LIN {X -112.913,Y -21.431,Z -236.404,A -90.000,B 90.000,C 0.000} C_DIS
LIN {X -101.773,Y -21.431,Z -228.606,A -90.000,B 90.000,C 0.000} C_DIS
LIN {X -97.009,Y -21.431,Z -225.268,A -90.000,B 90.000,C 0.000} C_DIS
LIN {X -92.221,Y -21.431,Z -221.963,A -90.000,B 90.000,C 0.000} C_DIS
LIN {X -87.411,Y -21.431,Z -218.691,A -90.000,B 90.000,C 0.000} C_DIS
LIN {X -82.578,Y -21.431,Z -215.452,A -90.000,B 90.000,C 0.000} C_DIS
LIN {X -77.723,Y -21.431,Z -212.248,A -90.000,B 90.000,C 0.000} C_DIS
LIN {X -69.739,Y -21.431,Z -206.990,A -90.000,B 90.000,C 0.000} C_DIS
LIN {X -65.801,Y -21.431,Z -204.457,A -90.000,B 90.000,C 0.000} C_DIS
LIN {X -61.895,Y -21.431,Z -201.875,A -90.000,B 90.000,C 0.000} C_DIS
LIN {X -58.021,Y -21.431,Z -199.246,A -90.000,B 90.000,C 0.000} C_DIS
LIN {X -54.179,Y -21.431,Z -196.569,A -90.000,B 90.000,C 0.000} C_DIS
LIN {X -50.371,Y -21.431,Z -193.845,A -90.000,B 90.000,C 0.000} C_DIS
LIN {X -46.597,Y -21.431,Z -191.074,A -90.000,B 90.000,C 0.000} C_DIS
LIN {X -42.857,Y -21.431,Z -188.257,A -90.000,B 90.000,C 0.000} C_DIS
LIN {X -39.152,Y -21.431,Z -185.394,A -90.000,B 90.000,C 0.000} C_DIS
LIN {X -35.482,Y -21.431,Z -182.486,A -90.000,B 90.000,C 0.000} C_DIS
LIN {X -33.831,Y -21.431,Z -181.236,A -90.000,B 90.000,C 0.000} C_DIS
LIN {X -32.219,Y -21.431,Z -179.937,A -90.000,B 90.000,C 0.000} C_DIS
LIN {X -30.645,Y -21.431,Z -178.592,A -90.000,B 90.000,C 0.000} C_DIS
LIN {X -29.112,Y -21.431,Z -177.200,A -90.000,B 90.000,C 0.000} C_DIS
LIN {X -27.621,Y -21.431,Z -175.763,A -90.000,B 90.000,C 0.000} C_DIS
LIN {X -26.173,Y -21.431,Z -174.283,A -90.000,B 90.000,C 0.000} C_DIS
LIN {X -24.770,Y -21.431,Z -172.761,A -90.000,B 90.000,C 0.000} C_DIS
LIN {X -23.815,Y -21.431,Z -171.758,A -90.000,B 90.000,C 0.000} C_DIS
LIN {X -22.906,Y -21.431,Z -170.713,A -90.000,B 90.000,C 0.000} C_DIS
LIN {X -22.045,Y -21.431,Z -169.628,A -90.000,B 90.000,C 0.000} C_DIS
LIN {X -21.234,Y -21.431,Z -168.506,A -90.000,B 90.000,C 0.000} C_DIS
LIN {X -20.473,Y -21.431,Z -167.349,A -90.000,B 90.000,C 0.000} C_DIS
LIN {X -19.766,Y -21.431,Z -166.158,A -90.000,B 90.000,C 0.000} C_DIS
LIN {X -19.112,Y -21.431,Z -164.937,A -90.000,B 90.000,C 0.000} C_DIS
LIN {X -18.514,Y -21.431,Z -163.688,A -90.000,B 90.000,C 0.000} C_DIS
LIN {X -18.456,Y -21.431,Z -163.541,A -90.000,B 90.000,C 0.000} C_DIS
LIN {X -19.036,Y -21.431,Z -162.884,A -90.000,B 90.000,C 0.000} C_DIS
LIN {X -19.116,Y -21.431,Z -162.777,A -90.000,B 90.000,C 0.000} C_DIS
LIN {X -19.886,Y -21.431,Z -161.971,A -90.000,B 90.000,C 0.000} C_DIS
LIN {X -20.688,Y -21.431,Z -161.196,A -90.000,B 90.000,C 0.000} C_DIS
LIN {X -23.607,Y -21.431,Z -158.546,A -90.000,B 90.000,C 0.000} C_DIS
LIN {X -26.501,Y -21.431,Z -155.871,A -90.000,B 90.000,C 0.000} C_DIS
LIN {X -29.372,Y -21.431,Z -153.169,A -90.000,B 90.000,C 0.000} C_DIS
LIN {X -30.672,Y -21.431,Z -151.944,A -90.000,B 90.000,C 0.000} C_DIS
LIN {X -31.934,Y -21.431,Z -150.679,A -90.000,B 90.000,C 0.000} C_DIS
LIN {X -33.157,Y -21.431,Z -149.377,A -90.000,B 90.000,C 0.000} C_DIS
LIN {X -34.339,Y -21.431,Z -148.039,A -90.000,B 90.000,C 0.000} C_DIS
LIN {X -35.481,Y -21.431,Z -146.664,A -90.000,B 90.000,C 0.000} C_DIS
LIN {X -36.579,Y -21.431,Z -145.256,A -90.000,B 90.000,C 0.000} C_DIS
LIN {X -37.635,Y -21.431,Z -143.815,A -90.000,B 90.000,C 0.000} C_DIS
LIN {X -38.762,Y -21.431,Z -142.053,A -90.000,B 90.000,C 0.000} C_DIS
LIN {X -39.842,Y -21.431,Z -140.263,A -90.000,B 90.000,C 0.000} C_DIS
LIN {X -40.874,Y -21.431,Z -138.445,A -90.000,B 90.000,C 0.000} C_DIS
LIN {X -41.859,Y -21.431,Z -136.600,A -90.000,B 90.000,C 0.000} C_DIS
LIN {X -42.796,Y -21.431,Z -134.730,A -90.000,B 90.000,C 0.000} C_DIS
LIN {X -43.682,Y -21.431,Z -132.837,A -90.000,B 90.000,C 0.000} C_DIS
LIN {X -44.519,Y -21.431,Z -130.920,A -90.000,B 90.000,C 0.000} C_DIS
LIN {X -45.306,Y -21.431,Z -128.983,A -90.000,B 90.000,C 0.000} C_DIS
LIN {X -45.631,Y -21.431,Z -127.972,A -90.000,B 90.000,C 0.000} C_DIS
LIN {X -46.007,Y -21.431,Z -126.979,A -90.000,B 90.000,C 0.000} C_DIS
LIN {X -46.431,Y -21.431,Z -126.006,A -90.000,B 90.000,C 0.000} C_DIS
LIN {X -46.904,Y -21.431,Z -125.055,A -90.000,B 90.000,C 0.000} C_DIS
LIN {X -47.424,Y -21.431,Z -124.129,A -90.000,B 90.000,C 0.000} C_DIS
LIN {X -47.989,Y -21.431,Z -123.230,A -90.000,B 90.000,C 0.000} C_DIS
LIN {X -50.279,Y -21.431,Z -120.489,A -90.000,B 90.000,C 0.000} C_DIS
LIN {X -52.532,Y -21.431,Z -117.717,A -90.000,B 90.000,C 0.000} C_DIS
LIN {X -54.746,Y -21.431,Z -114.914,A -90.000,B 90.000,C 0.000} C_DIS
LIN {X -56.921,Y -21.431,Z -112.081,A -90.000,B 90.000,C 0.000} C_DIS
LIN {X -59.058,Y -21.431,Z -109.218,A -90.000,B 90.000,C 0.000} C_DIS
LIN {X -61.154,Y -21.431,Z -106.326,A -90.000,B 90.000,C 0.000} C_DIS
LIN {X -62.757,Y -21.431,Z -104.098,A -90.000,B 90.000,C 0.000} C_DIS
LIN {X -64.383,Y -21.431,Z -101.888,A -90.000,B 90.000,C 0.000} C_DIS
LIN {X -65.729,Y -21.431,Z -100.052,A -90.000,B 90.000,C 0.000} C_DIS
LIN {X -67.124,Y -21.431,Z -98.251,A -90.000,B 90.000,C 0.000} C_DIS
LIN {X -68.566,Y -21.431,Z -96.489,A -90.000,B 90.000,C 0.000} C_DIS
LIN {X -70.054,Y -21.431,Z -94.765,A -90.000,B 90.000,C 0.000} C_DIS
LIN {X -71.588,Y -21.431,Z -93.082,A -90.000,B 90.000,C 0.000} C_DIS
LIN {X -73.165,Y -21.431,Z -91.439,A -90.000,B 90.000,C 0.000} C_DIS
LIN {X -74.786,Y -21.431,Z -89.839,A -90.000,B 90.000,C 0.000} C_DIS
LIN {X -76.448,Y -21.431,Z -88.283,A -90.000,B 90.000,C 0.000} C_DIS
LIN {X -76.915,Y -21.431,Z -87.802,A -90.000,B 90.000,C 0.000} C_DIS
LIN {X -77.417,Y -21.431,Z -87.357,A -90.000,B 90.000,C 0.000} C_DIS
LIN {X -77.950,Y -21.431,Z -86.950,A -90.000,B 90.000,C 0.000} C_DIS
LIN {X -78.511,Y -21.431,Z -86.584,A -90.000,B 90.000,C 0.000} C_DIS
LIN {X -79.099,Y -21.431,Z -86.260,A -90.000,B 90.000,C 0.000} C_DIS
LIN {X -79.708,Y -21.431,Z -85.980,A -90.000,B 90.000,C 0.000} C_DIS
LIN {X -81.105,Y -21.431,Z -85.489,A -90.000,B 90.000,C 0.000} C_DIS
LIN {X -82.479,Y -21.431,Z -84.936,A -90.000,B 90.000,C 0.000} C_DIS
LIN {X -83.828,Y -21.431,Z -84.323,A -90.000,B 90.000,C 0.000} C_DIS
LIN {X -85.147,Y -21.431,Z -83.651,A -90.000,B 90.000,C 0.000} C_DIS
LIN {X -86.436,Y -21.431,Z -82.921,A -90.000,B 90.000,C 0.000} C_DIS
LIN {X -87.691,Y -21.431,Z -82.134,A -90.000,B 90.000,C 0.000} C_DIS
LIN {X -88.909,Y -21.431,Z -81.292,A -90.000,B 90.000,C 0.000} C_DIS
LIN {X -90.090,Y -21.431,Z -80.398,A -90.000,B 90.000,C 0.000} C_DIS
LIN {X -90.244,Y -21.431,Z -80.288,A -90.000,B 90.000,C 0.000} C_DIS
LIN {X -92.608,Y -21.431,Z -78.373,A -90.000,B 90.000,C 0.000} C_DIS
LIN {X -94.982,Y -21.431,Z -76.470,A -90.000,B 90.000,C 0.000} C_DIS
LIN {X -96.724,Y -21.431,Z -75.460,A -90.000,B 90.000,C 0.000} C_DIS
LIN {X -98.431,Y -21.431,Z -74.393,A -90.000,B 90.000,C 0.000} C_DIS
LIN {X -100.102,Y -21.431,Z -73.269,A -90.000,B 90.000,C 0.000} C_DIS
LIN {X -101.734,Y -21.431,Z -72.091,A -90.000,B 90.000,C 0.000} C_DIS
LIN {X -103.327,Y -21.431,Z -70.859,A -90.000,B 90.000,C 0.000} C_DIS
LIN {X -104.877,Y -21.431,Z -69.575,A -90.000,B 90.000,C 0.000} C_DIS
LIN {X -106.385,Y -21.431,Z -68.240,A -90.000,B 90.000,C 0.000} C_DIS
LIN {X -107.846,Y -21.431,Z -66.856,A -90.000,B 90.000,C 0.000} C_DIS
LIN {X -109.262,Y -21.431,Z -65.424,A -90.000,B 90.000,C 0.000} C_DIS
LIN {X -110.628,Y -21.431,Z -63.945,A -90.000,B 90.000,C 0.000} C_DIS
LIN {X -111.945,Y -21.431,Z -62.422,A -90.000,B 90.000,C 0.000} C_DIS
LIN {X -112.631,Y -21.431,Z -61.641,A -90.000,B 90.000,C 0.000} C_DIS
LIN {X -113.269,Y -21.431,Z -60.819,A -90.000,B 90.000,C 0.000} C_DIS
LIN {X -113.855,Y -21.431,Z -59.960,A -90.000,B 90.000,C 0.000} C_DIS
LIN {X -114.388,Y -21.431,Z -59.066,A -90.000,B 90.000,C 0.000} C_DIS
LIN {X -114.865,Y -21.431,Z -58.142,A -90.000,B 90.000,C 0.000} C_DIS
LIN {X -115.284,Y -21.431,Z -57.190,A -90.000,B 90.000,C 0.000} C_DIS
LIN {X -115.645,Y -21.431,Z -56.215,A -90.000,B 90.000,C 0.000} C_DIS
LIN {X -115.945,Y -21.431,Z -55.219,A -90.000,B 90.000,C 0.000} C_DIS
LIN {X -116.219,Y -21.431,Z -54.365,A -90.000,B 90.000,C 0.000} C_DIS
LIN {X -116.430,Y -21.431,Z -53.494,A -90.000,B 90.000,C 0.000} C_DIS
LIN {X -116.579,Y -21.431,Z -52.609,A -90.000,B 90.000,C 0.000} C_DIS
LIN {X -116.664,Y -21.431,Z -51.717,A -90.000,B 90.000,C 0.000} C_DIS
LIN {X -116.684,Y -21.431,Z -50.820,A -90.000,B 90.000,C 0.000} C_DIS
LIN {X -116.640,Y -21.431,Z -49.924,A -90.000,B 90.000,C 0.000} C_DIS
LIN {X -116.532,Y -21.431,Z -49.034,A -90.000,B 90.000,C 0.000} C_DIS
LIN {X -116.361,Y -21.431,Z -48.154,A -90.000,B 90.000,C 0.000} C_DIS
LIN {X -116.729,Y -21.431,Z -47.203,A -90.000,B 90.000,C 0.000} C_DIS
LIN {X -117.034,Y -21.431,Z -46.230,A -90.000,B 90.000,C 0.000} C_DIS
LIN {X -117.276,Y -21.431,Z -45.239,A -90.000,B 90.000,C 0.000} C_DIS
LIN {X -117.453,Y -21.431,Z -44.235,A -90.000,B 90.000,C 0.000} C_DIS
LIN {X -117.565,Y -21.431,Z -43.221,A -90.000,B 90.000,C 0.000} C_DIS
LIN {X -117.611,Y -21.431,Z -42.203,A -90.000,B 90.000,C 0.000} C_DIS
LIN {X -117.592,Y -21.431,Z -41.183,A -90.000,B 90.000,C 0.000} C_DIS
LIN {X -117.506,Y -21.431,Z -40.167,A -90.000,B 90.000,C 0.000} C_DIS
LIN {X -117.481,Y -21.431,Z -39.998,A -90.000,B 90.000,C 0.000} C_DIS
LIN {X -117.325,Y -21.431,Z -39.111,A -90.000,B 90.000,C 0.000} C_DIS
LIN {X -117.112,Y -21.431,Z -38.236,A -90.000,B 90.000,C 0.000} C_DIS
LIN {X -116.843,Y -21.431,Z -37.377,A -90.000,B 90.000,C 0.000} C_DIS
LIN {X -116.518,Y -21.431,Z -36.537,A -90.000,B 90.000,C 0.000} C_DIS
LIN {X -116.140,Y -21.431,Z -35.720,A -90.000,B 90.000,C 0.000} C_DIS
LIN {X -115.709,Y -21.431,Z -34.929,A -90.000,B 90.000,C 0.000} C_DIS
LIN {X -115.632,Y -21.431,Z -34.808,A -90.000,B 90.000,C 0.000} C_DIS
LIN {X -115.195,Y -21.431,Z -34.136,A -90.000,B 90.000,C 0.000} C_DIS
LIN {X -114.713,Y -21.431,Z -33.495,A -90.000,B 90.000,C 0.000} C_DIS
LIN {X -114.188,Y -21.431,Z -32.888,A -90.000,B 90.000,C 0.000} C_DIS
LIN {X -113.624,Y -21.431,Z -32.318,A -90.000,B 90.000,C 0.000} C_DIS
LIN {X -113.490,Y -21.431,Z -32.194,A -90.000,B 90.000,C 0.000} C_DIS
LIN {X -112.360,Y -21.431,Z -31.268,A -90.000,B 90.000,C 0.000} C_DIS
LIN {X -112.270,Y -21.431,Z -31.206,A -90.000,B 90.000,C 0.000} C_DIS
LIN {X -111.804,Y -21.431,Z -30.880,A -90.000,B 90.000,C 0.000} C_DIS
LIN {X -111.318,Y -21.431,Z -30.585,A -90.000,B 90.000,C 0.000} C_DIS
LIN {X -110.813,Y -21.431,Z -30.324,A -90.000,B 90.000,C 0.000} C_DIS
LIN {X -110.292,Y -21.431,Z -30.095,A -90.000,B 90.000,C 0.000} C_DIS
LIN {X -109.345,Y -21.431,Z -29.251,A -90.000,B 90.000,C 0.000} C_DIS
LIN {X -108.357,Y -21.431,Z -28.456,A -90.000,B 90.000,C 0.000} C_DIS
LIN {X -107.331,Y -21.431,Z -27.711,A -90.000,B 90.000,C 0.000} C_DIS
LIN {X -106.268,Y -21.431,Z -27.018,A -90.000,B 90.000,C 0.000} C_DIS
LIN {X -105.172,Y -21.431,Z -26.380,A -90.000,B 90.000,C 0.000} C_DIS
LIN {X -104.800,Y -21.431,Z -25.659,A -90.000,B 90.000,C 0.000} C_DIS
LIN {X -104.385,Y -21.431,Z -24.961,A -90.000,B 90.000,C 0.000} C_DIS
LIN {X -103.928,Y -21.431,Z -24.289,A -90.000,B 90.000,C 0.000} C_DIS
LIN {X -103.432,Y -21.431,Z -23.647,A -90.000,B 90.000,C 0.000} C_DIS
LIN {X -102.917,Y -21.431,Z -22.919,A -90.000,B 90.000,C 0.000} C_DIS
LIN {X -102.353,Y -21.431,Z -22.229,A -90.000,B 90.000,C 0.000} C_DIS
LIN {X -101.741,Y -21.431,Z -21.581,A -90.000,B 90.000,C 0.000} C_DIS
LIN {X -101.084,Y -21.431,Z -20.977,A -90.000,B 90.000,C 0.000} C_DIS
LIN {X -100.387,Y -21.431,Z -20.422,A -90.000,B 90.000,C 0.000} C_DIS
LIN {X -99.653,Y -21.431,Z -19.917,A -90.000,B 90.000,C 0.000} C_DIS
LIN {X -98.884,Y -21.431,Z -19.465,A -90.000,B 90.000,C 0.000} C_DIS
LIN {X -98.086,Y -21.431,Z -19.068,A -90.000,B 90.000,C 0.000} C_DIS
LIN {X -97.261,Y -21.431,Z -18.729,A -90.000,B 90.000,C 0.000} C_DIS
LIN {X -96.126,Y -21.431,Z -18.440,A -90.000,B 90.000,C 0.000} C_DIS
LIN {X -94.976,Y -21.431,Z -18.214,A -90.000,B 90.000,C 0.000} C_DIS
LIN {X -93.816,Y -21.431,Z -18.051,A -90.000,B 90.000,C 0.000} C_DIS
LIN {X -92.649,Y -21.431,Z -17.952,A -90.000,B 90.000,C 0.000} C_DIS
LIN {X -91.478,Y -21.431,Z -17.916,A -90.000,B 90.000,C 0.000} C_DIS
LIN {X -91.153,Y -21.431,Z -17.123,A -90.000,B 90.000,C 0.000} C_DIS
LIN {X -90.777,Y -21.431,Z -16.352,A -90.000,B 90.000,C 0.000} C_DIS
LIN {X -90.350,Y -21.431,Z -15.609,A -90.000,B 90.000,C 0.000} C_DIS
LIN {X -89.876,Y -21.431,Z -14.895,A -90.000,B 90.000,C 0.000} C_DIS
LIN {X -89.355,Y -21.431,Z -14.214,A -90.000,B 90.000,C 0.000} C_DIS
LIN {X -88.791,Y -21.431,Z -13.568,A -90.000,B 90.000,C 0.000} C_DIS
LIN {X -88.035,Y -21.431,Z -12.875,A -90.000,B 90.000,C 0.000} C_DIS
LIN {X -87.234,Y -21.431,Z -12.236,A -90.000,B 90.000,C 0.000} C_DIS
LIN {X -86.391,Y -21.431,Z -11.651,A -90.000,B 90.000,C 0.000} C_DIS
LIN {X -85.512,Y -21.431,Z -11.125,A -90.000,B 90.000,C 0.000} C_DIS
LIN {X -84.598,Y -21.431,Z -10.660,A -90.000,B 90.000,C 0.000} C_DIS
LIN {X -83.655,Y -21.431,Z -10.257,A -90.000,B 90.000,C 0.000} C_DIS
LIN {X -82.687,Y -21.431,Z -9.919,A -90.000,B 90.000,C 0.000} C_DIS
LIN {X -81.699,Y -21.431,Z -9.647,A -90.000,B 90.000,C 0.000} C_DIS
LIN {X -80.694,Y -21.431,Z -9.442,A -90.000,B 90.000,C 0.000} C_DIS
LIN {X -79.678,Y -21.431,Z -9.306,A -90.000,B 90.000,C 0.000} C_DIS
LIN {X -78.655,Y -21.431,Z -9.238,A -90.000,B 90.000,C 0.000} C_DIS
LIN {X -77.406,Y -21.431,Z -9.311,A -90.000,B 90.000,C 0.000} C_DIS
LIN {X -76.163,Y -21.431,Z -9.451,A -90.000,B 90.000,C 0.000} C_DIS
LIN {X -74.929,Y -21.431,Z -9.660,A -90.000,B 90.000,C 0.000} C_DIS
LIN {X -73.709,Y -21.431,Z -9.935,A -90.000,B 90.000,C 0.000} C_DIS
LIN {X -72.505,Y -21.431,Z -10.276,A -90.000,B 90.000,C 0.000} C_DIS
LIN {X -71.322,Y -21.431,Z -10.683,A -90.000,B 90.000,C 0.000} C_DIS
LIN {X -70.163,Y -21.431,Z -11.153,A -90.000,B 90.000,C 0.000} C_DIS
LIN {X -69.031,Y -21.431,Z -11.687,A -90.000,B 90.000,C 0.000} C_DIS
LIN {X -67.874,Y -21.431,Z -12.293,A -90.000,B 90.000,C 0.000} C_DIS
LIN {X -66.751,Y -21.431,Z -12.959,A -90.000,B 90.000,C 0.000} C_DIS
LIN {X -65.664,Y -21.431,Z -13.684,A -90.000,B 90.000,C 0.000} C_DIS
LIN {X -64.617,Y -21.431,Z -14.465,A -90.000,B 90.000,C 0.000} C_DIS
LIN {X -63.613,Y -21.431,Z -15.300,A -90.000,B 90.000,C 0.000} C_DIS
LIN {X -62.655,Y -21.431,Z -16.188,A -90.000,B 90.000,C 0.000} C_DIS
LIN {X -61.745,Y -21.431,Z -17.124,A -90.000,B 90.000,C 0.000} C_DIS
LIN {X -60.885,Y -21.431,Z -18.107,A -90.000,B 90.000,C 0.000} C_DIS
LIN {X -60.078,Y -21.431,Z -19.135,A -90.000,B 90.000,C 0.000} C_DIS
LIN {X -59.327,Y -21.431,Z -20.203,A -90.000,B 90.000,C 0.000} C_DIS
LIN {X -58.595,Y -21.431,Z -21.635,A -90.000,B 90.000,C 0.000} C_DIS
LIN {X -57.857,Y -21.431,Z -23.063,A -90.000,B 90.000,C 0.000} C_DIS
LIN {X -57.794,Y -21.431,Z -23.212,A -90.000,B 90.000,C 0.000} C_DIS
LIN {X -56.492,Y -21.431,Z -23.608,A -90.000,B 90.000,C 0.000} C_DIS
LIN {X -55.174,Y -21.431,Z -23.948,A -90.000,B 90.000,C 0.000} C_DIS
LIN {X -53.842,Y -21.431,Z -24.230,A -90.000,B 90.000,C 0.000} C_DIS
LIN {X -52.500,Y -21.431,Z -24.455,A -90.000,B 90.000,C 0.000} C_DIS
LIN {X -51.149,Y -21.431,Z -24.621,A -90.000,B 90.000,C 0.000} C_DIS
LIN {X -49.792,Y -21.431,Z -24.728,A -90.000,B 90.000,C 0.000} C_DIS
LIN {X -49.617,Y -21.431,Z -24.736,A -90.000,B 90.000,C 0.000} C_DIS
LIN {X -48.809,Y -21.431,Z -24.706,A -90.000,B 90.000,C 0.000} C_DIS
LIN {X -48.001,Y -21.431,Z -24.720,A -90.000,B 90.000,C 0.000} C_DIS
LIN {X -47.195,Y -21.431,Z -24.779,A -90.000,B 90.000,C 0.000} C_DIS
LIN {X -46.393,Y -21.431,Z -24.883,A -90.000,B 90.000,C 0.000} C_DIS
LIN {X -43.339,Y -21.431,Z -24.939,A -90.000,B 90.000,C 0.000} C_DIS
LIN {X -40.286,Y -21.431,Z -25.061,A -90.000,B 90.000,C 0.000} C_DIS
LIN {X -37.237,Y -21.431,Z -25.249,A -90.000,B 90.000,C 0.000} C_DIS
LIN {X -34.193,Y -21.431,Z -25.503,A -90.000,B 90.000,C 0.000} C_DIS
LIN {X -31.155,Y -21.431,Z -25.823,A -90.000,B 90.000,C 0.000} C_DIS
LIN {X -28.125,Y -21.431,Z -26.209,A -90.000,B 90.000,C 0.000} C_DIS
LIN {X -25.104,Y -21.431,Z -26.660,A -90.000,B 90.000,C 0.000} C_DIS
LIN {X -22.093,Y -21.431,Z -27.176,A -90.000,B 90.000,C 0.000} C_DIS
LIN {X -19.094,Y -21.431,Z -27.758,A -90.000,B 90.000,C 0.000} C_DIS
LIN {X -16.108,Y -21.431,Z -28.404,A -90.000,B 90.000,C 0.000} C_DIS
LIN {X -13.137,Y -21.431,Z -29.114,A -90.000,B 90.000,C 0.000} C_DIS
LIN {X -10.182,Y -21.431,Z -29.889,A -90.000,B 90.000,C 0.000} C_DIS
LIN {X -7.245,Y -21.431,Z -30.728,A -90.000,B 90.000,C 0.000} C_DIS
LIN {X -6.078,Y -21.431,Z -31.125,A -90.000,B 90.000,C 0.000} C_DIS
LIN {X -4.894,Y -21.431,Z -31.466,A -90.000,B 90.000,C 0.000} C_DIS
LIN {X -3.694,Y -21.431,Z -31.750,A -90.000,B 90.000,C 0.000} C_DIS
LIN {X -2.482,Y -21.431,Z -31.977,A -90.000,B 90.000,C 0.000} C_DIS
LIN {X -1.261,Y -21.431,Z -32.145,A -90.000,B 90.000,C 0.000} C_DIS
LIN {X -0.034,Y -21.431,Z -32.255,A -90.000,B 90.000,C 0.000} C_DIS
LIN {X 1.198,Y -21.431,Z -32.305,A -90.000,B 90.000,C 0.000} C_DIS
LIN {X 3.136,Y -21.431,Z -32.301,A -90.000,B 90.000,C 0.000} C_DIS
LIN {X 5.073,Y -21.431,Z -32.346,A -90.000,B 90.000,C 0.000} C_DIS
LIN {X 7.009,Y -21.431,Z -32.440,A -90.000,B 90.000,C 0.000} C_DIS
LIN {X 8.942,Y -21.431,Z -32.584,A -90.000,B 90.000,C 0.000} C_DIS
LIN {X 10.870,Y -21.431,Z -32.776,A -90.000,B 90.000,C 0.000} C_DIS
LIN {X 12.793,Y -21.431,Z -33.017,A -90.000,B 90.000,C 0.000} C_DIS
LIN {X 14.148,Y -21.431,Z -33.216,A -90.000,B 90.000,C 0.000} C_DIS
LIN {X 15.510,Y -21.431,Z -33.360,A -90.000,B 90.000,C 0.000} C_DIS
LIN {X 16.877,Y -21.431,Z -33.450,A -90.000,B 90.000,C 0.000} C_DIS
LIN {X 18.246,Y -21.431,Z -33.486,A -90.000,B 90.000,C 0.000} C_DIS
LIN {X 19.616,Y -21.431,Z -33.466,A -90.000,B 90.000,C 0.000} C_DIS
LIN {X 20.983,Y -21.431,Z -33.392,A -90.000,B 90.000,C 0.000} C_DIS
LIN {X 22.347,Y -21.431,Z -33.264,A -90.000,B 90.000,C 0.000} C_DIS
LIN {X 25.111,Y -21.431,Z -32.751,A -90.000,B 90.000,C 0.000} C_DIS
LIN {X 27.884,Y -21.431,Z -32.288,A -90.000,B 90.000,C 0.000} C_DIS
LIN {X 30.665,Y -21.431,Z -31.876,A -90.000,B 90.000,C 0.000} C_DIS
LIN {X 33.453,Y -21.431,Z -31.514,A -90.000,B 90.000,C 0.000} C_DIS
LIN {X 35.088,Y -21.431,Z -31.430,A -90.000,B 90.000,C 0.000} C_DIS
LIN {X 36.726,Y -21.431,Z -31.411,A -90.000,B 90.000,C 0.000} C_DIS
LIN {X 38.362,Y -21.431,Z -31.456,A -90.000,B 90.000,C 0.000} C_DIS
LIN {X 39.996,Y -21.431,Z -31.566,A -90.000,B 90.000,C 0.000} C_DIS
LIN {X 41.624,Y -21.431,Z -31.741,A -90.000,B 90.000,C 0.000} C_DIS
LIN {X 43.244,Y -21.431,Z -31.980,A -90.000,B 90.000,C 0.000} C_DIS
LIN {X 44.853,Y -21.431,Z -32.283,A -90.000,B 90.000,C 0.000} C_DIS
LIN {X 46.520,Y -21.431,Z -32.778,A -90.000,B 90.000,C 0.000} C_DIS
LIN {X 48.167,Y -21.431,Z -33.333,A -90.000,B 90.000,C 0.000} C_DIS
LIN {X 49.794,Y -21.431,Z -33.947,A -90.000,B 90.000,C 0.000} C_DIS
LIN {X 51.397,Y -21.431,Z -34.619,A -90.000,B 90.000,C 0.000} C_DIS
LIN {X 52.976,Y -21.431,Z -35.348,A -90.000,B 90.000,C 0.000} C_DIS
LIN {X 54.527,Y -21.431,Z -36.133,A -90.000,B 90.000,C 0.000} C_DIS
LIN {X 56.049,Y -21.431,Z -36.974,A -90.000,B 90.000,C 0.000} C_DIS
LIN {X 57.539,Y -21.431,Z -37.869,A -90.000,B 90.000,C 0.000} C_DIS
LIN {X 58.997,Y -21.431,Z -38.817,A -90.000,B 90.000,C 0.000} C_DIS
LIN {X 60.419,Y -21.431,Z -39.816,A -90.000,B 90.000,C 0.000} C_DIS
LIN {X 61.805,Y -21.431,Z -40.866,A -90.000,B 90.000,C 0.000} C_DIS
LIN {X 62.842,Y -21.431,Z -41.828,A -90.000,B 90.000,C 0.000} C_DIS
LIN {X 63.911,Y -21.431,Z -42.753,A -90.000,B 90.000,C 0.000} C_DIS
LIN {X 65.011,Y -21.431,Z -43.642,A -90.000,B 90.000,C 0.000} C_DIS
LIN {X 66.140,Y -21.431,Z -44.494,A -90.000,B 90.000,C 0.000} C_DIS
LIN {X 67.298,Y -21.431,Z -45.306,A -90.000,B 90.000,C 0.000} C_DIS
LIN {X 68.482,Y -21.431,Z -46.079,A -90.000,B 90.000,C 0.000} C_DIS
LIN {X 70.165,Y -21.431,Z -46.968,A -90.000,B 90.000,C 0.000} C_DIS
LIN {X 71.828,Y -21.431,Z -47.895,A -90.000,B 90.000,C 0.000} C_DIS
LIN {X 73.468,Y -21.431,Z -48.860,A -90.000,B 90.000,C 0.000} C_DIS
LIN {X 75.086,Y -21.431,Z -49.863,A -90.000,B 90.000,C 0.000} C_DIS
LIN {X 76.681,Y -21.431,Z -50.902,A -90.000,B 90.000,C 0.000} C_DIS
LIN {X 77.484,Y -21.431,Z -49.408,A -90.000,B 90.000,C 0.000} C_DIS
LIN {X 78.417,Y -21.431,Z -47.991,A -90.000,B 90.000,C 0.000} C_DIS
LIN {X 79.409,Y -21.431,Z -46.615,A -90.000,B 90.000,C 0.000} C_DIS
LIN {X 80.458,Y -21.431,Z -45.282,A -90.000,B 90.000,C 0.000} C_DIS
LIN {X 81.563,Y -21.431,Z -43.995,A -90.000,B 90.000,C 0.000} C_DIS
LIN {X 82.722,Y -21.431,Z -42.757,A -90.000,B 90.000,C 0.000} C_DIS
LIN {X 83.933,Y -21.431,Z -41.568,A -90.000,B 90.000,C 0.000} C_DIS
LIN {X 85.193,Y -21.431,Z -40.433,A -90.000,B 90.000,C 0.000} C_DIS
LIN {X 86.500,Y -21.431,Z -39.351,A -90.000,B 90.000,C 0.000} C_DIS
LIN {X 87.852,Y -21.431,Z -38.327,A -90.000,B 90.000,C 0.000} C_DIS
LIN {X 89.246,Y -21.431,Z -37.360,A -90.000,B 90.000,C 0.000} C_DIS
LIN {X 91.067,Y -21.431,Z -36.216,A -90.000,B 90.000,C 0.000} C_DIS
LIN {X 92.918,Y -21.431,Z -35.121,A -90.000,B 90.000,C 0.000} C_DIS
LIN {X 94.797,Y -21.431,Z -34.076,A -90.000,B 90.000,C 0.000} C_DIS
LIN {X 96.704,Y -21.431,Z -33.081,A -90.000,B 90.000,C 0.000} C_DIS
LIN {X 98.636,Y -21.431,Z -32.137,A -90.000,B 90.000,C 0.000} C_DIS
LIN {X 100.592,Y -21.431,Z -31.245,A -90.000,B 90.000,C 0.000} C_DIS
LIN {X 102.572,Y -21.431,Z -30.405,A -90.000,B 90.000,C 0.000} C_DIS
LIN {X 104.573,Y -21.431,Z -29.618,A -90.000,B 90.000,C 0.000} C_DIS
LIN {X 105.513,Y -21.431,Z -29.233,A -90.000,B 90.000,C 0.000} C_DIS
LIN {X 106.478,Y -21.431,Z -28.915,A -90.000,B 90.000,C 0.000} C_DIS
LIN {X 107.464,Y -21.431,Z -28.667,A -90.000,B 90.000,C 0.000} C_DIS
LIN {X 108.464,Y -21.431,Z -28.489,A -90.000,B 90.000,C 0.000} C_DIS
LIN {X 109.474,Y -21.431,Z -28.382,A -90.000,B 90.000,C 0.000} C_DIS
LIN {X 110.490,Y -21.431,Z -28.346,A -90.000,B 90.000,C 0.000} C_DIS
LIN {X 111.505,Y -21.431,Z -28.383,A -90.000,B 90.000,C 0.000} C_DIS
LIN {X 112.516,Y -21.431,Z -28.492,A -90.000,B 90.000,C 0.000} C_DIS
LIN {X 113.516,Y -21.431,Z -28.671,A -90.000,B 90.000,C 0.000} C_DIS
LIN {X 114.501,Y -21.431,Z -28.921,A -90.000,B 90.000,C 0.000} C_DIS
LIN {X 115.465,Y -21.431,Z -29.240,A -90.000,B 90.000,C 0.000} C_DIS
LIN {X 116.405,Y -21.431,Z -29.627,A -90.000,B 90.000,C 0.000} C_DIS
LIN {X 117.315,Y -21.431,Z -30.079,A -90.000,B 90.000,C 0.000} C_DIS
LIN {X 118.191,Y -21.431,Z -30.594,A -90.000,B 90.000,C 0.000} C_DIS
LIN {X 119.028,Y -21.431,Z -31.170,A -90.000,B 90.000,C 0.000} C_DIS
LIN {X 119.134,Y -21.431,Z -31.254,A -90.000,B 90.000,C 0.000} C_DIS
LIN {X 119.816,Y -21.431,Z -31.834,A -90.000,B 90.000,C 0.000} C_DIS
LIN {X 120.465,Y -21.431,Z -32.450,A -90.000,B 90.000,C 0.000} C_DIS
LIN {X 121.081,Y -21.431,Z -33.099,A -90.000,B 90.000,C 0.000} C_DIS
LIN {X 121.662,Y -21.431,Z -33.780,A -90.000,B 90.000,C 0.000} C_DIS
LIN {X 122.196,Y -21.431,Z -34.612,A -90.000,B 90.000,C 0.000} C_DIS
LIN {X 122.676,Y -21.431,Z -35.476,A -90.000,B 90.000,C 0.000} C_DIS
LIN {X 123.102,Y -21.431,Z -36.368,A -90.000,B 90.000,C 0.000} C_DIS
LIN {X 123.470,Y -21.431,Z -37.286,A -90.000,B 90.000,C 0.000} C_DIS
LIN {X 123.781,Y -21.431,Z -38.224,A -90.000,B 90.000,C 0.000} C_DIS
LIN {X 124.032,Y -21.431,Z -39.180,A -90.000,B 90.000,C 0.000} C_DIS
LIN {X 124.222,Y -21.431,Z -40.150,A -90.000,B 90.000,C 0.000} C_DIS
LIN {X 124.352,Y -21.431,Z -41.130,A -90.000,B 90.000,C 0.000} C_DIS
LIN {X 124.419,Y -21.431,Z -42.117,A -90.000,B 90.000,C 0.000} C_DIS
LIN {X 124.425,Y -21.431,Z -43.105,A -90.000,B 90.000,C 0.000} C_DIS
LIN {X 124.369,Y -21.431,Z -44.092,A -90.000,B 90.000,C 0.000} C_DIS
LIN {X 124.170,Y -21.431,Z -45.366,A -90.000,B 90.000,C 0.000} C_DIS
LIN {X 123.911,Y -21.431,Z -46.630,A -90.000,B 90.000,C 0.000} C_DIS
LIN {X 123.595,Y -21.431,Z -47.880,A -90.000,B 90.000,C 0.000} C_DIS
LIN {X 123.220,Y -21.431,Z -49.114,A -90.000,B 90.000,C 0.000} C_DIS
LIN {X 122.789,Y -21.431,Z -50.330,A -90.000,B 90.000,C 0.000} C_DIS
LIN {X 122.302,Y -21.431,Z -51.524,A -90.000,B 90.000,C 0.000} C_DIS
LIN {X 121.760,Y -21.431,Z -52.694,A -90.000,B 90.000,C 0.000} C_DIS
LIN {X 121.061,Y -21.431,Z -53.939,A -90.000,B 90.000,C 0.000} C_DIS
LIN {X 120.409,Y -21.431,Z -55.208,A -90.000,B 90.000,C 0.000} C_DIS
LIN {X 119.804,Y -21.431,Z -56.501,A -90.000,B 90.000,C 0.000} C_DIS
LIN {X 119.247,Y -21.431,Z -57.815,A -90.000,B 90.000,C 0.000} C_DIS
LIN {X 118.739,Y -21.431,Z -59.149,A -90.000,B 90.000,C 0.000} C_DIS
LIN {X 118.281,Y -21.431,Z -60.500,A -90.000,B 90.000,C 0.000} C_DIS
LIN {X 117.872,Y -21.431,Z -61.868,A -90.000,B 90.000,C 0.000} C_DIS
LIN {X 117.358,Y -21.431,Z -63.979,A -90.000,B 90.000,C 0.000} C_DIS
LIN {X 116.784,Y -21.431,Z -66.075,A -90.000,B 90.000,C 0.000} C_DIS
LIN {X 116.150,Y -21.431,Z -68.153,A -90.000,B 90.000,C 0.000} C_DIS
LIN {X 115.456,Y -21.431,Z -70.212,A -90.000,B 90.000,C 0.000} C_DIS
LIN {X 114.703,Y -21.431,Z -72.250,A -90.000,B 90.000,C 0.000} C_DIS
LIN {X 113.892,Y -21.431,Z -74.265,A -90.000,B 90.000,C 0.000} C_DIS
LIN {X 113.023,Y -21.431,Z -76.257,A -90.000,B 90.000,C 0.000} C_DIS
LIN {X 112.096,Y -21.431,Z -78.222,A -90.000,B 90.000,C 0.000} C_DIS
LIN {X 111.114,Y -21.431,Z -80.160,A -90.000,B 90.000,C 0.000} C_DIS
LIN {X 110.076,Y -21.431,Z -82.069,A -90.000,B 90.000,C 0.000} C_DIS
LIN {X 108.984,Y -21.431,Z -83.947,A -90.000,B 90.000,C 0.000} C_DIS
LIN {X 107.838,Y -21.431,Z -85.793,A -90.000,B 90.000,C 0.000} C_DIS
LIN {X 106.639,Y -21.431,Z -87.605,A -90.000,B 90.000,C 0.000} C_DIS
LIN {X 106.699,Y -21.431,Z -88.459,A -90.000,B 90.000,C 0.000} C_DIS
LIN {X 107.090,Y -21.431,Z -89.542,A -90.000,B 90.000,C 0.000} C_DIS
LIN {X 107.424,Y -21.431,Z -90.644,A -90.000,B 90.000,C 0.000} C_DIS
LIN {X 107.700,Y -21.431,Z -91.761,A -90.000,B 90.000,C 0.000} C_DIS
LIN {X 107.917,Y -21.431,Z -92.892,A -90.000,B 90.000,C 0.000} C_DIS
LIN {X 107.942,Y -21.431,Z -93.067,A -90.000,B 90.000,C 0.000} C_DIS
LIN {X 108.302,Y -21.431,Z -95.300,A -90.000,B 90.000,C 0.000} C_DIS
LIN {X 108.631,Y -21.431,Z -97.537,A -90.000,B 90.000,C 0.000} C_DIS
LIN {X 108.638,Y -21.431,Z -97.630,A -90.000,B 90.000,C 0.000} C_DIS
LIN {X 108.827,Y -21.431,Z -98.875,A -90.000,B 90.000,C 0.000} C_DIS
LIN {X 108.843,Y -21.431,Z -99.059,A -90.000,B 90.000,C 0.000} C_DIS
LIN {X 109.069,Y -21.431,Z -100.622,A -90.000,B 90.000,C 0.000} C_DIS
LIN {X 109.313,Y -21.431,Z -102.183,A -90.000,B 90.000,C 0.000} C_DIS
LIN {X 109.880,Y -21.431,Z -105.571,A -90.000,B 90.000,C 0.000} C_DIS
LIN {X 110.389,Y -21.431,Z -108.969,A -90.000,B 90.000,C 0.000} C_DIS
LIN {X 110.841,Y -21.431,Z -112.375,A -90.000,B 90.000,C 0.000} C_DIS
LIN {X 111.235,Y -21.431,Z -115.788,A -90.000,B 90.000,C 0.000} C_DIS
LIN {X 111.571,Y -21.431,Z -119.207,A -90.000,B 90.000,C 0.000} C_DIS
LIN {X 111.850,Y -21.431,Z -122.631,A -90.000,B 90.000,C 0.000} C_DIS
LIN {X 112.070,Y -21.431,Z -126.059,A -90.000,B 90.000,C 0.000} C_DIS
LIN {X 112.232,Y -21.431,Z -129.491,A -90.000,B 90.000,C 0.000} C_DIS
LIN {X 112.216,Y -21.431,Z -133.540,A -90.000,B 90.000,C 0.000} C_DIS
LIN {X 112.146,Y -21.431,Z -137.588,A -90.000,B 90.000,C 0.000} C_DIS
LIN {X 112.021,Y -21.431,Z -141.635,A -90.000,B 90.000,C 0.000} C_DIS
LIN {X 111.843,Y -21.431,Z -145.680,A -90.000,B 90.000,C 0.000} C_DIS
LIN {X 111.611,Y -21.431,Z -149.722,A -90.000,B 90.000,C 0.000} C_DIS
LIN {X 111.325,Y -21.431,Z -153.760,A -90.000,B 90.000,C 0.000} C_DIS
LIN {X 110.985,Y -21.431,Z -157.795,A -90.000,B 90.000,C 0.000} C_DIS
LIN {X 110.574,Y -21.431,Z -162.937,A -90.000,B 90.000,C 0.000} C_DIS
LIN {X 110.090,Y -21.431,Z -168.072,A -90.000,B 90.000,C 0.000} C_DIS
LIN {X 109.536,Y -21.431,Z -173.201,A -90.000,B 90.000,C 0.000} C_DIS
LIN {X 108.909,Y -21.431,Z -178.321,A -90.000,B 90.000,C 0.000} C_DIS
LIN {X 108.211,Y -21.431,Z -183.432,A -90.000,B 90.000,C 0.000} C_DIS
LIN {X 107.441,Y -21.431,Z -188.532,A -90.000,B 90.000,C 0.000} C_DIS
LIN {X 106.601,Y -21.431,Z -193.621,A -90.000,B 90.000,C 0.000} C_DIS
LIN {X 105.689,Y -21.431,Z -198.698,A -90.000,B 90.000,C 0.000} C_DIS
LIN {X 104.706,Y -21.431,Z -203.762,A -90.000,B 90.000,C 0.000} C_DIS
LIN {X 103.653,Y -21.431,Z -208.812,A -90.000,B 90.000,C 0.000} C_DIS
LIN {X 102.529,Y -21.431,Z -213.846,A -90.000,B 90.000,C 0.000} C_DIS
LIN {X 101.334,Y -21.431,Z -218.864,A -90.000,B 90.000,C 0.000} C_DIS
LIN {X 100.506,Y -21.431,Z -222.436,A -90.000,B 90.000,C 0.000} C_DIS
LIN {X 99.622,Y -21.431,Z -225.995,A -90.000,B 90.000,C 0.000} C_DIS
LIN {X 98.683,Y -21.431,Z -229.540,A -90.000,B 90.000,C 0.000} C_DIS
LIN {X 97.689,Y -21.431,Z -233.070,A -90.000,B 90.000,C 0.000} C_DIS
LIN {X 96.641,Y -21.431,Z -236.584,A -90.000,B 90.000,C 0.000} C_DIS
LIN {X 95.537,Y -21.431,Z -240.081,A -90.000,B 90.000,C 0.000} C_DIS
LIN {X 94.380,Y -21.431,Z -243.561,A -90.000,B 90.000,C 0.000} C_DIS
LIN {X 145.015,Y -21.431,Z -243.561,A -90.000,B 90.000,C 0.000} C_DIS
LIN {X 145.015,Y -33.931,Z -243.561,A -90.000,B 90.000,C 0.000} C_DIS
LIN {X 145.015,Y -46.431,Z -243.561,A -90.000,B 90.000,C 0.000} C_DIS
LIN {X 145.015,Y -57.084,Z -243.561,A -90.000,B 90.000,C 0.000} C_DIS
LIN {X -144.015,Y -57.084,Z -242.561,A -90.000,B 90.000,C 0.000} C_DIS
LIN {X -144.015,Y -39.288,Z -242.561,A -90.000,B 90.000,C 0.000} C_DIS
LIN {X -144.015,Y -26.788,Z -242.561,A -90.000,B 90.000,C 0.000} C_DIS
LIN {X -144.015,Y -14.287,Z -242.561,A -90.000,B 90.000,C 0.000} C_DIS
LIN {X -137.090,Y -14.287,Z -242.561,A -90.000,B 90.000,C 0.000} C_DIS
LIN {X -136.812,Y -14.287,Z -242.289,A -90.000,B 90.000,C 0.000} C_DIS
LIN {X -134.866,Y -14.287,Z -240.849,A -90.000,B 90.000,C 0.000} C_DIS
LIN {X -132.892,Y -14.287,Z -239.450,A -90.000,B 90.000,C 0.000} C_DIS
LIN {X -130.889,Y -14.287,Z -238.091,A -90.000,B 90.000,C 0.000} C_DIS
LIN {X -128.859,Y -14.287,Z -236.773,A -90.000,B 90.000,C 0.000} C_DIS
LIN {X -126.317,Y -14.287,Z -235.012,A -90.000,B 90.000,C 0.000} C_DIS
LIN {X -144.015,Y -14.287,Z -235.012,A -90.000,B 90.000,C 0.000} C_DIS
LIN {X -144.015,Y -14.287,Z -227.464,A -90.000,B 90.000,C 0.000} C_DIS
LIN {X -115.194,Y -14.287,Z -227.464,A -90.000,B 90.000,C 0.000} C_DIS
LIN {X -111.375,Y -14.287,Z -224.928,A -90.000,B 90.000,C 0.000} C_DIS
LIN {X -107.543,Y -14.287,Z -222.412,A -90.000,B 90.000,C 0.000} C_DIS
LIN {X -103.698,Y -14.287,Z -219.915,A -90.000,B 90.000,C 0.000} C_DIS
LIN {X -144.015,Y -14.287,Z -219.915,A -90.000,B 90.000,C 0.000} C_DIS
LIN {X -144.015,Y -14.287,Z -212.366,A -90.000,B 90.000,C 0.000} C_DIS
LIN {X -91.801,Y -14.287,Z -212.366,A -90.000,B 90.000,C 0.000} C_DIS
LIN {X -87.192,Y -14.287,Z -209.512,A -90.000,B 90.000,C 0.000} C_DIS
LIN {X -82.565,Y -14.287,Z -206.685,A -90.000,B 90.000,C 0.000} C_DIS
LIN {X -79.476,Y -14.287,Z -204.817,A -90.000,B 90.000,C 0.000} C_DIS
LIN {X -144.015,Y -14.287,Z -204.817,A -90.000,B 90.000,C 0.000} C_DIS
LIN {X -144.015,Y -14.287,Z -197.269,A -90.000,B 90.000,C 0.000} C_DIS
LIN {X -66.930,Y -14.287,Z -197.269,A -90.000,B 90.000,C 0.000} C_DIS
LIN {X -65.753,Y -14.287,Z -196.570,A -90.000,B 90.000,C 0.000} C_DIS
LIN {X -62.889,Y -14.287,Z -194.912,A -90.000,B 90.000,C 0.000} C_DIS
LIN {X -60.046,Y -14.287,Z -193.218,A -90.000,B 90.000,C 0.000} C_DIS
LIN {X -57.225,Y -14.287,Z -191.487,A -90.000,B 90.000,C 0.000} C_DIS
LIN {X -54.426,Y -14.287,Z -189.720,A -90.000,B 90.000,C 0.000} C_DIS
LIN {X -144.015,Y -14.287,Z -189.720,A -90.000,B 90.000,C 0.000} C_DIS
LIN {X -144.015,Y -14.287,Z -182.171,A -90.000,B 90.000,C 0.000} C_DIS
LIN {X -43.292,Y -14.287,Z -182.171,A -90.000,B 90.000,C 0.000} C_DIS
LIN {X -41.154,Y -14.287,Z -180.621,A -90.000,B 90.000,C 0.000} C_DIS
LIN {X -39.031,Y -14.287,Z -179.050,A -90.000,B 90.000,C 0.000} C_DIS
LIN {X -37.579,Y -14.287,Z -177.998,A -90.000,B 90.000,C 0.000} C_DIS
LIN {X -36.154,Y -14.287,Z -176.909,A -90.000,B 90.000,C 0.000} C_DIS
LIN {X -34.758,Y -14.287,Z -175.783,A -90.000,B 90.000,C 0.000} C_DIS
LIN {X -33.392,Y -14.287,Z -174.622,A -90.000,B 90.000,C 0.000} C_DIS
LIN {X -144.015,Y -14.287,Z -174.622,A -90.000,B 90.000,C 0.000} C_DIS
LIN {X -144.015,Y -14.287,Z -167.073,A -90.000,B 90.000,C 0.000} C_DIS
LIN {X -26.264,Y -14.287,Z -167.073,A -90.000,B 90.000,C 0.000} C_DIS
LIN {X -25.590,Y -14.287,Z -166.025,A -90.000,B 90.000,C 0.000} C_DIS
LIN {X -24.966,Y -14.287,Z -164.945,A -90.000,B 90.000,C 0.000} C_DIS
LIN {X -24.395,Y -14.287,Z -163.837,A -90.000,B 90.000,C 0.000} C_DIS
LIN {X -23.876,Y -14.287,Z -162.704,A -90.000,B 90.000,C 0.000} C_DIS
LIN {X -24.228,Y -14.287,Z -162.207,A -90.000,B 90.000,C 0.000} C_DIS
LIN {X -24.609,Y -14.287,Z -161.733,A -90.000,B 90.000,C 0.000} C_DIS
LIN {X -26.734,Y -14.287,Z -159.525,A -90.000,B 90.000,C 0.000} C_DIS
LIN {X -144.015,Y -14.287,Z -159.525,A -90.000,B 90.000,C 0.000} C_DIS
LIN {X -144.015,Y -14.287,Z -151.976,A -90.000,B 90.000,C 0.000} C_DIS
LIN {X -34.074,Y -14.287,Z -151.976,A -90.000,B 90.000,C 0.000} C_DIS
LIN {X -35.228,Y -14.287,Z -150.666,A -90.000,B 90.000,C 0.000} C_DIS
LIN {X -36.347,Y -14.287,Z -149.325,A -90.000,B 90.000,C 0.000} C_DIS
LIN {X -37.429,Y -14.287,Z -147.955,A -90.000,B 90.000,C 0.000} C_DIS
LIN {X -38.474,Y -14.287,Z -146.557,A -90.000,B 90.000,C 0.000} C_DIS
LIN {X -39.481,Y -14.287,Z -145.130,A -90.000,B 90.000,C 0.000} C_DIS
LIN {X -39.925,Y -14.287,Z -144.427,A -90.000,B 90.000,C 0.000} C_DIS
LIN {X -144.015,Y -14.287,Z -144.427,A -90.000,B 90.000,C 0.000} C_DIS
LIN {X -144.015,Y -14.287,Z -136.878,A -90.000,B 90.000,C 0.000} C_DIS
LIN {X -44.194,Y -14.287,Z -136.878,A -90.000,B 90.000,C 0.000} C_DIS
LIN {X -45.117,Y -14.287,Z -135.018,A -90.000,B 90.000,C 0.000} C_DIS
LIN {X -46.001,Y -14.287,Z -133.140,A -90.000,B 90.000,C 0.000} C_DIS
LIN {X -46.846,Y -14.287,Z -131.243,A -90.000,B 90.000,C 0.000} C_DIS
LIN {X -47.651,Y -14.287,Z -129.329,A -90.000,B 90.000,C 0.000} C_DIS
LIN {X -144.015,Y -14.287,Z -129.329,A -90.000,B 90.000,C 0.000} C_DIS
LIN {X -144.015,Y -14.287,Z -121.781,A -90.000,B 90.000,C 0.000} C_DIS
LIN {X -52.023,Y -14.287,Z -121.781,A -90.000,B 90.000,C 0.000} C_DIS
LIN {X -54.072,Y -14.287,Z -119.287,A -90.000,B 90.000,C 0.000} C_DIS
LIN {X -56.093,Y -14.287,Z -116.770,A -90.000,B 90.000,C 0.000} C_DIS
LIN {X -58.087,Y -14.287,Z -114.232,A -90.000,B 90.000,C 0.000} C_DIS
LIN {X -144.015,Y -14.287,Z -114.232,A -90.000,B 90.000,C 0.000} C_DIS
LIN {X -144.015,Y -14.287,Z -106.683,A -90.000,B 90.000,C 0.000} C_DIS
LIN {X -63.747,Y -14.287,Z -106.683,A -90.000,B 90.000,C 0.000} C_DIS
LIN {X -64.714,Y -14.287,Z -105.352,A -90.000,B 90.000,C 0.000} C_DIS
LIN {X -65.718,Y -14.287,Z -104.049,A -90.000,B 90.000,C 0.000} C_DIS
LIN {X -66.759,Y -14.287,Z -102.774,A -90.000,B 90.000,C 0.000} C_DIS
LIN {X -67.835,Y -14.287,Z -101.530,A -90.000,B 90.000,C 0.000} C_DIS
LIN {X -68.946,Y -14.287,Z -100.316,A -90.000,B 90.000,C 0.000} C_DIS
LIN {X -70.090,Y -14.287,Z -99.134,A -90.000,B 90.000,C 0.000} C_DIS
LIN {X -144.015,Y -14.287,Z -99.134,A -90.000,B 90.000,C 0.000} C_DIS
LIN {X -144.015,Y -14.287,Z -91.586,A -90.000,B 90.000,C 0.000} C_DIS
LIN {X -80.163,Y -14.287,Z -91.586,A -90.000,B 90.000,C 0.000} C_DIS
LIN {X -80.249,Y -14.287,Z -91.531,A -90.000,B 90.000,C 0.000} C_DIS
LIN {X -81.724,Y -14.287,Z -90.672,A -90.000,B 90.000,C 0.000} C_DIS
LIN {X -83.174,Y -14.287,Z -89.769,A -90.000,B 90.000,C 0.000} C_DIS
LIN {X -84.596,Y -14.287,Z -88.824,A -90.000,B 90.000,C 0.000} C_DIS
LIN {X -85.989,Y -14.287,Z -87.837,A -90.000,B 90.000,C 0.000} C_DIS
LIN {X -87.353,Y -14.287,Z -86.810,A -90.000,B 90.000,C 0.000} C_DIS
LIN {X -88.686,Y -14.287,Z -85.742,A -90.000,B 90.000,C 0.000} C_DIS
LIN {X -89.987,Y -14.287,Z -84.637,A -90.000,B 90.000,C 0.000} C_DIS
LIN {X -90.258,Y -14.287,Z -84.330,A -90.000,B 90.000,C 0.000} C_DIS
LIN {X -90.545,Y -14.287,Z -84.037,A -90.000,B 90.000,C 0.000} C_DIS
LIN {X -144.015,Y -14.287,Z -84.037,A -90.000,B 90.000,C 0.000} C_DIS
LIN {X -144.015,Y -14.287,Z -76.488,A -90.000,B 90.000,C 0.000} C_DIS
LIN {X -109.086,Y -14.287,Z -76.488,A -90.000,B 90.000,C 0.000} C_DIS
LIN {X -110.171,Y -14.287,Z -75.526,A -90.000,B 90.000,C 0.000} C_DIS
LIN {X -111.218,Y -14.287,Z -74.522,A -90.000,B 90.000,C 0.000} C_DIS
LIN {X -112.224,Y -14.287,Z -73.479,A -90.000,B 90.000,C 0.000} C_DIS
LIN {X -113.190,Y -14.287,Z -72.397,A -90.000,B 90.000,C 0.000} C_DIS
LIN {X -114.113,Y -14.287,Z -71.279,A -90.000,B 90.000,C 0.000} C_DIS
LIN {X -114.992,Y -14.287,Z -70.126,A -90.000,B 90.000,C 0.000} C_DIS
LIN {X -115.825,Y -14.287,Z -68.939,A -90.000,B 90.000,C 0.000} C_DIS
LIN {X -144.015,Y -14.287,Z -68.939,A -90.000,B 90.000,C 0.000} C_DIS
LIN {X -144.015,Y -14.287,Z -61.390,A -90.000,B 90.000,C 0.000} C_DIS
LIN {X -119.527,Y -14.287,Z -61.390,A -90.000,B 90.000,C 0.000} C_DIS
LIN {X -119.973,Y -14.287,Z -59.927,A -90.000,B 90.000,C 0.000} C_DIS
LIN {X -120.370,Y -14.287,Z -58.449,A -90.000,B 90.000,C 0.000} C_DIS
LIN {X -120.716,Y -14.287,Z -56.959,A -90.000,B 90.000,C 0.000} C_DIS
LIN {X -121.019,Y -14.287,Z -56.201,A -90.000,B 90.000,C 0.000} C_DIS
LIN {X -121.279,Y -14.287,Z -55.427,A -90.000,B 90.000,C 0.000} C_DIS
LIN {X -121.496,Y -14.287,Z -54.640,A -90.000,B 90.000,C 0.000} C_DIS
LIN {X -121.668,Y -14.287,Z -53.842,A -90.000,B 90.000,C 0.000} C_DIS
LIN {X -144.015,Y -14.287,Z -53.842,A -90.000,B 90.000,C 0.000} C_DIS
LIN {X -144.015,Y -14.287,Z -46.293,A -90.000,B 90.000,C 0.000} C_DIS
LIN {X -123.293,Y -14.287,Z -46.293,A -90.000,B 90.000,C 0.000} C_DIS
LIN {X -123.257,Y -14.287,Z -45.575,A -90.000,B 90.000,C 0.000} C_DIS
LIN {X -123.185,Y -14.287,Z -44.861,A -90.000,B 90.000,C 0.000} C_DIS
LIN {X -123.075,Y -14.287,Z -44.150,A -90.000,B 90.000,C 0.000} C_DIS
LIN {X -122.928,Y -14.287,Z -43.447,A -90.000,B 90.000,C 0.000} C_DIS
LIN {X -123.246,Y -14.287,Z -42.533,A -90.000,B 90.000,C 0.000} C_DIS
LIN {X -123.512,Y -14.287,Z -41.603,A -90.000,B 90.000,C 0.000} C_DIS
LIN {X -123.725,Y -14.287,Z -40.660,A -90.000,B 90.000,C 0.000} C_DIS
LIN {X -123.885,Y -14.287,Z -39.706,A -90.000,B 90.000,C 0.000} C_DIS
LIN {X -123.990,Y -14.287,Z -38.744,A -90.000,B 90.000,C 0.000} C_DIS
LIN {X -144.015,Y -14.287,Z -38.744,A -90.000,B 90.000,C 0.000} C_DIS
LIN {X -144.015,Y -14.287,Z -31.195,A -90.000,B 90.000,C 0.000} C_DIS
LIN {X -122.928,Y -14.287,Z -31.195,A -90.000,B 90.000,C 0.000} C_DIS
LIN {X -122.596,Y -14.287,Z -30.351,A -90.000,B 90.000,C 0.000} C_DIS
LIN {X -122.209,Y -14.287,Z -29.530,A -90.000,B 90.000,C 0.000} C_DIS
LIN {X -121.769,Y -14.287,Z -28.737,A -90.000,B 90.000,C 0.000} C_DIS
LIN {X -121.277,Y -14.287,Z -27.975,A -90.000,B 90.000,C 0.000} C_DIS
LIN {X -120.735,Y -14.287,Z -27.247,A -90.000,B 90.000,C 0.000} C_DIS
LIN {X -120.146,Y -14.287,Z -26.557,A -90.000,B 90.000,C 0.000} C_DIS
LIN {X -119.512,Y -14.287,Z -25.908,A -90.000,B 90.000,C 0.000} C_DIS
LIN {X -118.983,Y -14.287,Z -25.130,A -90.000,B 90.000,C 0.000} C_DIS
LIN {X -118.421,Y -14.287,Z -24.375,A -90.000,B 90.000,C 0.000} C_DIS
LIN {X -117.826,Y -14.287,Z -23.646,A -90.000,B 90.000,C 0.000} C_DIS
LIN {X -144.015,Y -14.287,Z -23.646,A -90.000,B 90.000,C 0.000} C_DIS
LIN {X -144.015,Y -14.287,Z -16.098,A -90.000,B 90.000,C 0.000} C_DIS
LIN {X -106.610,Y -14.287,Z -16.098,A -90.000,B 90.000,C 0.000} C_DIS
LIN {X -106.563,Y -14.287,Z -16.040,A -90.000,B 90.000,C 0.000} C_DIS
LIN {X -106.474,Y -14.287,Z -15.947,A -90.000,B 90.000,C 0.000} C_DIS
LIN {X -105.854,Y -14.287,Z -15.336,A -90.000,B 90.000,C 0.000} C_DIS
LIN {X -105.194,Y -14.287,Z -14.767,A -90.000,B 90.000,C 0.000} C_DIS
LIN {X -104.499,Y -14.287,Z -14.243,A -90.000,B 90.000,C 0.000} C_DIS
LIN {X -103.771,Y -14.287,Z -13.765,A -90.000,B 90.000,C 0.000} C_DIS
LIN {X -103.351,Y -14.287,Z -13.580,A -90.000,B 90.000,C 0.000} C_DIS
LIN {X -102.953,Y -14.287,Z -13.350,A -90.000,B 90.000,C 0.000} C_DIS
LIN {X -102.584,Y -14.287,Z -13.077,A -90.000,B 90.000,C 0.000} C_DIS
LIN {X -102.476,Y -14.287,Z -12.982,A -90.000,B 90.000,C 0.000} C_DIS
LIN {X -101.703,Y -14.287,Z -12.322,A -90.000,B 90.000,C 0.000} C_DIS
LIN {X -100.899,Y -14.287,Z -11.699,A -90.000,B 90.000,C 0.000} C_DIS
LIN {X -100.065,Y -14.287,Z -11.117,A -90.000,B 90.000,C 0.000} C_DIS
LIN {X -99.205,Y -14.287,Z -10.576,A -90.000,B 90.000,C 0.000} C_DIS
LIN {X -98.318,Y -14.287,Z -10.078,A -90.000,B 90.000,C 0.000} C_DIS
LIN {X -97.409,Y -14.287,Z -9.623,A -90.000,B 90.000,C 0.000} C_DIS
LIN {X -97.243,Y -14.287,Z -9.555,A -90.000,B 90.000,C 0.000} C_DIS
LIN {X -96.183,Y -14.287,Z -9.167,A -90.000,B 90.000,C 0.000} C_DIS
LIN {X -95.105,Y -14.287,Z -8.831,A -90.000,B 90.000,C 0.000} C_DIS
LIN {X -94.012,Y -14.287,Z -8.549,A -90.000,B 90.000,C 0.000} C_DIS
LIN {X -144.015,Y -14.287,Z -8.549,A -90.000,B 90.000,C 0.000} C_DIS
LIN {X -144.015,Y -14.287,Z -1.000,A -90.000,B 90.000,C 0.000} C_DIS
LIN {X 144.015,Y -14.287,Z -1.000,A -90.000,B 90.000,C 0.000} C_DIS
LIN {X 144.015,Y -14.287,Z -8.549,A -90.000,B 90.000,C 0.000} C_DIS
LIN {X -66.989,Y -14.287,Z -8.549,A -90.000,B 90.000,C 0.000} C_DIS
LIN {X -64.892,Y -14.287,Z -9.490,A -90.000,B 90.000,C 0.000} C_DIS
LIN {X -62.779,Y -14.287,Z -10.393,A -90.000,B 90.000,C 0.000} C_DIS
LIN {X -61.672,Y -14.287,Z -10.942,A -90.000,B 90.000,C 0.000} C_DIS
LIN {X -60.538,Y -14.287,Z -11.433,A -90.000,B 90.000,C 0.000} C_DIS
LIN {X -59.381,Y -14.287,Z -11.867,A -90.000,B 90.000,C 0.000} C_DIS
LIN {X -58.203,Y -14.287,Z -12.241,A -90.000,B 90.000,C 0.000} C_DIS
LIN {X -57.008,Y -14.287,Z -12.555,A -90.000,B 90.000,C 0.000} C_DIS
LIN {X -55.798,Y -14.287,Z -12.808,A -90.000,B 90.000,C 0.000} C_DIS
LIN {X -54.577,Y -14.287,Z -12.999,A -90.000,B 90.000,C 0.000} C_DIS
LIN {X -53.348,Y -14.287,Z -13.128,A -90.000,B 90.000,C 0.000} C_DIS
LIN {X -51.076,Y -14.287,Z -13.501,A -90.000,B 90.000,C 0.000} C_DIS
LIN {X -48.799,Y -14.287,Z -13.840,A -90.000,B 90.000,C 0.000} C_DIS
LIN {X -46.517,Y -14.287,Z -14.145,A -90.000,B 90.000,C 0.000} C_DIS
LIN {X -44.231,Y -14.287,Z -14.415,A -90.000,B 90.000,C 0.000} C_DIS
LIN {X -42.365,Y -14.287,Z -14.547,A -90.000,B 90.000,C 0.000} C_DIS
LIN {X -40.503,Y -14.287,Z -14.724,A -90.000,B 90.000,C 0.000} C_DIS
LIN {X -38.645,Y -14.287,Z -14.947,A -90.000,B 90.000,C 0.000} C_DIS
LIN {X -36.794,Y -14.287,Z -15.214,A -90.000,B 90.000,C 0.000} C_DIS
LIN {X -34.949,Y -14.287,Z -15.526,A -90.000,B 90.000,C 0.000} C_DIS
LIN {X -33.113,Y -14.287,Z -15.883,A -90.000,B 90.000,C 0.000} C_DIS
LIN {X -31.948,Y -14.287,Z -16.098,A -90.000,B 90.000,C 0.000} C_DIS
LIN {X 144.015,Y -14.287,Z -16.098,A -90.000,B 90.000,C 0.000} C_DIS
LIN {X 144.015,Y -14.287,Z -23.646,A -90.000,B 90.000,C 0.000} C_DIS
LIN {X 5.796,Y -14.287,Z -23.646,A -90.000,B 90.000,C 0.000} C_DIS
LIN {X 7.253,Y -14.287,Z -23.924,A -90.000,B 90.000,C 0.000} C_DIS
LIN {X 18.701,Y -14.287,Z -26.105,A -90.000,B 90.000,C 0.000} C_DIS
LIN {X 19.413,Y -14.287,Z -26.107,A -90.000,B 90.000,C 0.000} C_DIS
LIN {X 20.124,Y -14.287,Z -26.084,A -90.000,B 90.000,C 0.000} C_DIS
LIN {X 20.834,Y -14.287,Z -26.036,A -90.000,B 90.000,C 0.000} C_DIS
LIN {X 22.692,Y -14.287,Z -26.105,A -90.000,B 90.000,C 0.000} C_DIS
LIN {X 24.547,Y -14.287,Z -26.234,A -90.000,B 90.000,C 0.000} C_DIS
LIN {X 26.396,Y -14.287,Z -26.423,A -90.000,B 90.000,C 0.000} C_DIS
LIN {X 28.239,Y -14.287,Z -26.672,A -90.000,B 90.000,C 0.000} C_DIS
LIN {X 30.072,Y -14.287,Z -26.981,A -90.000,B 90.000,C 0.000} C_DIS
LIN {X 31.895,Y -14.287,Z -27.349,A -90.000,B 90.000,C 0.000} C_DIS
LIN {X 33.704,Y -14.287,Z -27.777,A -90.000,B 90.000,C 0.000} C_DIS
LIN {X 34.764,Y -14.287,Z -28.062,A -90.000,B 90.000,C 0.000} C_DIS
LIN {X 35.828,Y -14.287,Z -28.331,A -90.000,B 90.000,C 0.000} C_DIS
LIN {X 39.403,Y -14.287,Z -29.434,A -90.000,B 90.000,C 0.000} C_DIS
LIN {X 42.986,Y -14.287,Z -30.514,A -90.000,B 90.000,C 0.000} C_DIS
LIN {X 44.204,Y -14.287,Z -30.840,A -90.000,B 90.000,C 0.000} C_DIS
LIN {X 45.413,Y -14.287,Z -31.195,A -90.000,B 90.000,C 0.000} C_DIS
LIN {X 98.289,Y -14.287,Z -31.195,A -90.000,B 90.000,C 0.000} C_DIS
LIN {X 96.315,Y -14.287,Z -32.157,A -90.000,B 90.000,C 0.000} C_DIS
LIN {X 94.368,Y -14.287,Z -33.171,A -90.000,B 90.000,C 0.000} C_DIS
LIN {X 92.448,Y -14.287,Z -34.238,A -90.000,B 90.000,C 0.000} C_DIS
LIN {X 90.558,Y -14.287,Z -35.355,A -90.000,B 90.000,C 0.000} C_DIS
LIN {X 88.699,Y -14.287,Z -36.523,A -90.000,B 90.000,C 0.000} C_DIS
LIN {X 87.663,Y -14.287,Z -37.232,A -90.000,B 90.000,C 0.000} C_DIS
LIN {X 86.649,Y -14.287,Z -37.972,A -90.000,B 90.000,C 0.000} C_DIS
LIN {X 85.658,Y -14.287,Z -38.744,A -90.000,B 90.000,C 0.000} C_DIS
LIN {X 60.643,Y -14.287,Z -38.744,A -90.000,B 90.000,C 0.000} C_DIS
LIN {X 61.581,Y -14.287,Z -39.433,A -90.000,B 90.000,C 0.000} C_DIS
LIN {X 62.503,Y -14.287,Z -40.143,A -90.000,B 90.000,C 0.000} C_DIS
LIN {X 62.704,Y -14.287,Z -40.360,A -90.000,B 90.000,C 0.000} C_DIS
LIN {X 62.932,Y -14.287,Z -40.547,A -90.000,B 90.000,C 0.000} C_DIS
LIN {X 63.183,Y -14.287,Z -40.702,A -90.000,B 90.000,C 0.000} C_DIS
LIN {X 65.376,Y -14.287,Z -41.724,A -90.000,B 90.000,C 0.000} C_DIS
LIN {X 67.546,Y -14.287,Z -42.794,A -90.000,B 90.000,C 0.000} C_DIS
LIN {X 69.691,Y -14.287,Z -43.913,A -90.000,B 90.000,C 0.000} C_DIS
LIN {X 71.811,Y -14.287,Z -45.079,A -90.000,B 90.000,C 0.000} C_DIS
LIN {X 73.904,Y -14.287,Z -46.293,A -90.000,B 90.000,C 0.000} C_DIS
LIN {X 78.413,Y -14.287,Z -46.293,A -90.000,B 90.000,C 0.000} C_DIS
LIN {X 79.379,Y -14.287,Z -45.037,A -90.000,B 90.000,C 0.000} C_DIS
LIN {X 80.392,Y -14.287,Z -43.819,A -90.000,B 90.000,C 0.000} C_DIS
LIN {X 81.453,Y -14.287,Z -42.642,A -90.000,B 90.000,C 0.000} C_DIS
LIN {X 82.558,Y -14.287,Z -41.507,A -90.000,B 90.000,C 0.000} C_DIS
LIN {X 83.707,Y -14.287,Z -40.416,A -90.000,B 90.000,C 0.000} C_DIS
LIN {X 84.897,Y -14.287,Z -39.371,A -90.000,B 90.000,C 0.000} C_DIS
LIN {X 86.127,Y -14.287,Z -38.372,A -90.000,B 90.000,C 0.000} C_DIS
LIN {X 87.395,Y -14.287,Z -37.422,A -90.000,B 90.000,C 0.000} C_DIS
LIN {X 88.699,Y -14.287,Z -36.523,A -90.000,B 90.000,C 0.000} C_DIS
LIN {X 90.539,Y -14.287,Z -35.367,A -90.000,B 90.000,C 0.000} C_DIS
LIN {X 92.409,Y -14.287,Z -34.261,A -90.000,B 90.000,C 0.000} C_DIS
LIN {X 94.308,Y -14.287,Z -33.204,A -90.000,B 90.000,C 0.000} C_DIS
LIN {X 96.234,Y -14.287,Z -32.198,A -90.000,B 90.000,C 0.000} C_DIS
LIN {X 98.186,Y -14.287,Z -31.244,A -90.000,B 90.000,C 0.000} C_DIS
LIN {X 100.163,Y -14.287,Z -30.341,A -90.000,B 90.000,C 0.000} C_DIS
LIN {X 102.163,Y -14.287,Z -29.492,A -90.000,B 90.000,C 0.000} C_DIS
LIN {X 104.185,Y -14.287,Z -28.696,A -90.000,B 90.000,C 0.000} C_DIS
LIN {X 105.139,Y -14.287,Z -28.292,A -90.000,B 90.000,C 0.000} C_DIS
LIN {X 106.118,Y -14.287,Z -27.955,A -90.000,B 90.000,C 0.000} C_DIS
LIN {X 107.119,Y -14.287,Z -27.686,A -90.000,B 90.000,C 0.000} C_DIS
LIN {X 108.135,Y -14.287,Z -27.487,A -90.000,B 90.000,C 0.000} C_DIS
LIN {X 109.163,Y -14.287,Z -27.358,A -90.000,B 90.000,C 0.000} C_DIS
LIN {X 110.197,Y -14.287,Z -27.300,A -90.000,B 90.000,C 0.000} C_DIS
LIN {X 111.233,Y -14.287,Z -27.314,A -90.000,B 90.000,C 0.000} C_DIS
LIN {X 112.265,Y -14.287,Z -27.399,A -90.000,B 90.000,C 0.000} C_DIS
LIN {X 113.289,Y -14.287,Z -27.555,A -90.000,B 90.000,C 0.000} C_DIS
LIN {X 114.300,Y -14.287,Z -27.781,A -90.000,B 90.000,C 0.000} C_DIS
LIN {X 115.293,Y -14.287,Z -28.075,A -90.000,B 90.000,C 0.000} C_DIS
LIN {X 116.263,Y -14.287,Z -28.438,A -90.000,B 90.000,C 0.000} C_DIS
LIN {X 117.206,Y -14.287,Z -28.867,A -90.000,B 90.000,C 0.000} C_DIS
LIN {X 118.118,Y -14.287,Z -29.359,A -90.000,B 90.000,C 0.000} C_DIS
LIN {X 118.993,Y -14.287,Z -29.913,A -90.000,B 90.000,C 0.000} C_DIS
LIN {X 119.828,Y -14.287,Z -30.527,A -90.000,B 90.000,C 0.000} C_DIS
LIN {X 120.619,Y -14.287,Z -31.195,A -90.000,B 90.000,C 0.000} C_DIS
LIN {X 144.015,Y -14.287,Z -31.195,A -90.000,B 90.000,C 0.000} C_DIS
LIN {X 144.015,Y -14.287,Z -38.744,A -90.000,B 90.000,C 0.000} C_DIS
LIN {X 124.956,Y -14.287,Z -38.744,A -90.000,B 90.000,C 0.000} C_DIS
LIN {X 125.148,Y -14.287,Z -39.640,A -90.000,B 90.000,C 0.000} C_DIS
LIN {X 125.291,Y -14.287,Z -40.545,A -90.000,B 90.000,C 0.000} C_DIS
LIN {X 125.384,Y -14.287,Z -41.456,A -90.000,B 90.000,C 0.000} C_DIS
LIN {X 125.427,Y -14.287,Z -42.371,A -90.000,B 90.000,C 0.000} C_DIS
LIN {X 125.420,Y -14.287,Z -43.288,A -90.000,B 90.000,C 0.000} C_DIS
LIN {X 125.363,Y -14.287,Z -44.202,A -90.000,B 90.000,C 0.000} C_DIS
LIN {X 125.205,Y -14.287,Z -45.251,A -90.000,B 90.000,C 0.000} C_DIS
LIN {X 125.008,Y -14.287,Z -46.293,A -90.000,B 90.000,C 0.000} C_DIS
LIN {X 144.015,Y -14.287,Z -46.293,A -90.000,B 90.000,C 0.000} C_DIS
LIN {X 144.015,Y -14.287,Z -53.842,A -90.000,B 90.000,C 0.000} C_DIS
LIN {X 122.255,Y -14.287,Z -53.842,A -90.000,B 90.000,C 0.000} C_DIS
LIN {X 121.608,Y -14.287,Z -55.049,A -90.000,B 90.000,C 0.000} C_DIS
LIN {X 121.005,Y -14.287,Z -56.278,A -90.000,B 90.000,C 0.000} C_DIS
LIN {X 120.448,Y -14.287,Z -57.529,A -90.000,B 90.000,C 0.000} C_DIS
LIN {X 119.936,Y -14.287,Z -58.799,A -90.000,B 90.000,C 0.000} C_DIS
LIN {X 119.470,Y -14.287,Z -60.086,A -90.000,B 90.000,C 0.000} C_DIS
LIN {X 119.052,Y -14.287,Z -61.390,A -90.000,B 90.000,C 0.000} C_DIS
LIN {X 144.015,Y -14.287,Z -61.390,A -90.000,B 90.000,C 0.000} C_DIS
LIN {X 144.015,Y -14.287,Z -68.939,A -90.000,B 90.000,C 0.000} C_DIS
LIN {X 116.963,Y -14.287,Z -68.939,A -90.000,B 90.000,C 0.000} C_DIS
LIN {X 116.308,Y -14.287,Z -70.855,A -90.000,B 90.000,C 0.000} C_DIS
LIN {X 115.602,Y -14.287,Z -72.753,A -90.000,B 90.000,C 0.000} C_DIS
LIN {X 114.844,Y -14.287,Z -74.631,A -90.000,B 90.000,C 0.000} C_DIS
LIN {X 114.036,Y -14.287,Z -76.488,A -90.000,B 90.000,C 0.000} C_DIS
LIN {X 144.015,Y -14.287,Z -76.488,A -90.000,B 90.000,C 0.000} C_DIS
LIN {X 144.015,Y -14.287,Z -84.037,A -90.000,B 90.000,C 0.000} C_DIS
LIN {X 110.098,Y -14.287,Z -84.037,A -90.000,B 90.000,C 0.000} C_DIS
LIN {X 109.657,Y -14.287,Z -84.768,A -90.000,B 90.000,C 0.000} C_DIS
LIN {X 109.207,Y -14.287,Z -85.494,A -90.000,B 90.000,C 0.000} C_DIS
LIN {X 109.727,Y -14.287,Z -86.499,A -90.000,B 90.000,C 0.000} C_DIS
LIN {X 110.209,Y -14.287,Z -87.524,A -90.000,B 90.000,C 0.000} C_DIS
LIN {X 110.651,Y -14.287,Z -88.566,A -90.000,B 90.000,C 0.000} C_DIS
LIN {X 111.053,Y -14.287,Z -89.625,A -90.000,B 90.000,C 0.000} C_DIS
LIN {X 111.414,Y -14.287,Z -90.698,A -90.000,B 90.000,C 0.000} C_DIS
LIN {X 111.640,Y -14.287,Z -91.586,A -90.000,B 90.000,C 0.000} C_DIS
LIN {X 144.015,Y -14.287,Z -91.586,A -90.000,B 90.000,C 0.000} C_DIS
LIN {X 144.015,Y -14.287,Z -99.134,A -90.000,B 90.000,C 0.000} C_DIS
LIN {X 113.374,Y -14.287,Z -99.134,A -90.000,B 90.000,C 0.000} C_DIS
LIN {X 113.879,Y -14.287,Z -101.644,A -90.000,B 90.000,C 0.000} C_DIS
LIN {X 114.350,Y -14.287,Z -104.160,A -90.000,B 90.000,C 0.000} C_DIS
LIN {X 114.787,Y -14.287,Z -106.683,A -90.000,B 90.000,C 0.000} C_DIS
LIN {X 144.015,Y -14.287,Z -106.683,A -90.000,B 90.000,C 0.000} C_DIS
LIN {X 144.015,Y -14.287,Z -114.232,A -90.000,B 90.000,C 0.000} C_DIS
LIN {X 115.885,Y -14.287,Z -114.232,A -90.000,B 90.000,C 0.000} C_DIS
LIN {X 116.182,Y -14.287,Z -116.745,A -90.000,B 90.000,C 0.000} C_DIS
LIN {X 116.446,Y -14.287,Z -119.261,A -90.000,B 90.000,C 0.000} C_DIS
LIN {X 116.676,Y -14.287,Z -121.781,A -90.000,B 90.000,C 0.000} C_DIS
LIN {X 144.015,Y -14.287,Z -121.781,A -90.000,B 90.000,C 0.000} C_DIS
LIN {X 144.015,Y -14.287,Z -129.329,A -90.000,B 90.000,C 0.000} C_DIS
LIN {X 117.162,Y -14.287,Z -129.329,A -90.000,B 90.000,C 0.000} C_DIS
LIN {X 117.257,Y -14.287,Z -131.844,A -90.000,B 90.000,C 0.000} C_DIS
LIN {X 117.318,Y -14.287,Z -134.361,A -90.000,B 90.000,C 0.000} C_DIS
LIN {X 117.345,Y -14.287,Z -136.878,A -90.000,B 90.000,C 0.000} C_DIS
LIN {X 144.015,Y -14.287,Z -136.878,A -90.000,B 90.000,C 0.000} C_DIS
LIN {X 144.015,Y -14.287,Z -144.427,A -90.000,B 90.000,C 0.000} C_DIS
LIN {X 117.227,Y -14.287,Z -144.427,A -90.000,B 90.000,C 0.000} C_DIS
LIN {X 117.136,Y -14.287,Z -146.621,A -90.000,B 90.000,C 0.000} C_DIS
LIN {X 117.020,Y -14.287,Z -148.813,A -90.000,B 90.000,C 0.000} C_DIS
LIN {X 116.902,Y -14.287,Z -150.395,A -90.000,B 90.000,C 0.000} C_DIS
LIN {X 116.779,Y -14.287,Z -151.976,A -90.000,B 90.000,C 0.000} C_DIS
LIN {X 144.015,Y -14.287,Z -151.976,A -90.000,B 90.000,C 0.000} C_DIS
LIN {X 144.015,Y -14.287,Z -159.525,A -90.000,B 90.000,C 0.000} C_DIS
LIN {X 116.120,Y -14.287,Z -159.525,A -90.000,B 90.000,C 0.000} C_DIS
LIN {X 115.747,Y -14.287,Z -163.300,A -90.000,B 90.000,C 0.000} C_DIS
LIN {X 115.345,Y -14.287,Z -167.073,A -90.000,B 90.000,C 0.000} C_DIS
LIN {X 144.015,Y -14.287,Z -167.073,A -90.000,B 90.000,C 0.000} C_DIS
LIN {X 144.015,Y -14.287,Z -174.622,A -90.000,B 90.000,C 0.000} C_DIS
LIN {X 114.451,Y -14.287,Z -174.622,A -90.000,B 90.000,C 0.000} C_DIS
LIN {X 113.960,Y -14.287,Z -178.398,A -90.000,B 90.000,C 0.000} C_DIS
LIN {X 113.439,Y -14.287,Z -182.171,A -90.000,B 90.000,C 0.000} C_DIS
LIN {X 144.015,Y -14.287,Z -182.171,A -90.000,B 90.000,C 0.000} C_DIS
LIN {X 144.015,Y -14.287,Z -189.720,A -90.000,B 90.000,C 0.000} C_DIS
LIN {X 112.308,Y -14.287,Z -189.720,A -90.000,B 90.000,C 0.000} C_DIS
LIN {X 111.697,Y -14.287,Z -193.497,A -90.000,B 90.000,C 0.000} C_DIS
LIN {X 111.057,Y -14.287,Z -197.269,A -90.000,B 90.000,C 0.000} C_DIS
LIN {X 144.015,Y -14.287,Z -197.269,A -90.000,B 90.000,C 0.000} C_DIS
LIN {X 144.015,Y -14.287,Z -204.817,A -90.000,B 90.000,C 0.000} C_DIS
LIN {X 109.685,Y -14.287,Z -204.817,A -90.000,B 90.000,C 0.000} C_DIS
LIN {X 109.417,Y -14.287,Z -206.221,A -90.000,B 90.000,C 0.000} C_DIS
LIN {X 108.856,Y -14.287,Z -209.297,A -90.000,B 90.000,C 0.000} C_DIS
LIN {X 108.259,Y -14.287,Z -212.366,A -90.000,B 90.000,C 0.000} C_DIS
LIN {X 144.015,Y -14.287,Z -212.366,A -90.000,B 90.000,C 0.000} C_DIS
LIN {X 144.015,Y -14.287,Z -219.915,A -90.000,B 90.000,C 0.000} C_DIS
LIN {X 106.627,Y -14.287,Z -219.915,A -90.000,B 90.000,C 0.000} C_DIS
LIN {X 106.029,Y -14.287,Z -222.438,A -90.000,B 90.000,C 0.000} C_DIS
LIN {X 105.406,Y -14.287,Z -224.954,A -90.000,B 90.000,C 0.000} C_DIS
LIN {X 104.758,Y -14.287,Z -227.464,A -90.000,B 90.000,C 0.000} C_DIS
LIN {X 144.015,Y -14.287,Z -227.464,A -90.000,B 90.000,C 0.000} C_DIS
LIN {X 144.015,Y -14.287,Z -235.012,A -90.000,B 90.000,C 0.000} C_DIS
LIN {X 102.649,Y -14.287,Z -235.012,A -90.000,B 90.000,C 0.000} C_DIS
LIN {X 101.889,Y -14.287,Z -237.536,A -90.000,B 90.000,C 0.000} C_DIS
LIN {X 101.103,Y -14.287,Z -240.053,A -90.000,B 90.000,C 0.000} C_DIS
LIN {X 100.292,Y -14.287,Z -242.561,A -90.000,B 90.000,C 0.000} C_DIS
LIN {X 144.015,Y -14.287,Z -242.561,A -90.000,B 90.000,C 0.000} C_DIS
LIN {X 145.015,Y -14.287,Z -243.561,A -90.000,B 90.000,C 0.000} C_DIS
LIN {X 145.015,Y -14.287,Z 0.000,A -90.000,B 90.000,C 0.000} C_DIS
LIN {X -145.015,Y -14.287,Z 0.000,A -90.000,B 90.000,C 0.000} C_DIS
LIN {X -145.015,Y -14.287,Z -243.561,A -90.000,B 90.000,C 0.000} C_DIS
LIN {X -136.682,Y -14.287,Z -243.561,A -90.000,B 90.000,C 0.000} C_DIS
LIN {X -136.159,Y -14.287,Z -243.049,A -90.000,B 90.000,C 0.000} C_DIS
LIN {X -134.237,Y -14.287,Z -241.629,A -90.000,B 90.000,C 0.000} C_DIS
LIN {X -132.287,Y -14.287,Z -240.248,A -90.000,B 90.000,C 0.000} C_DIS
LIN {X -130.310,Y -14.287,Z -238.906,A -90.000,B 90.000,C 0.000} C_DIS
LIN {X -128.305,Y -14.287,Z -237.606,A -90.000,B 90.000,C 0.000} C_DIS
LIN {X -122.626,Y -14.287,Z -233.692,A -90.000,B 90.000,C 0.000} C_DIS
LIN {X -116.917,Y -14.287,Z -229.822,A -90.000,B 90.000,C 0.000} C_DIS
LIN {X -111.178,Y -14.287,Z -225.996,A -90.000,B 90.000,C 0.000} C_DIS
LIN {X -105.409,Y -14.287,Z -222.215,A -90.000,B 90.000,C 0.000} C_DIS
LIN {X -99.611,Y -14.287,Z -218.479,A -90.000,B 90.000,C 0.000} C_DIS
LIN {X -93.785,Y -14.287,Z -214.788,A -90.000,B 90.000,C 0.000} C_DIS
LIN {X -87.930,Y -14.287,Z -211.142,A -90.000,B 90.000,C 0.000} C_DIS
LIN {X -82.047,Y -14.287,Z -207.541,A -90.000,B 90.000,C 0.000} C_DIS
LIN {X -75.197,Y -14.287,Z -203.398,A -90.000,B 90.000,C 0.000} C_DIS
LIN {X -73.032,Y -14.287,Z -202.103,A -90.000,B 90.000,C 0.000} C_DIS
LIN {X -69.147,Y -14.287,Z -199.758,A -90.000,B 90.000,C 0.000} C_DIS
LIN {X -65.250,Y -14.287,Z -197.435,A -90.000,B 90.000,C 0.000} C_DIS
LIN {X -61.783,Y -14.287,Z -195.422,A -90.000,B 90.000,C 0.000} C_DIS
LIN {X -58.347,Y -14.287,Z -193.355,A -90.000,B 90.000,C 0.000} C_DIS
LIN {X -54.944,Y -14.287,Z -191.236,A -90.000,B 90.000,C 0.000} C_DIS
LIN {X -51.574,Y -14.287,Z -189.063,A -90.000,B 90.000,C 0.000} C_DIS
LIN {X -48.238,Y -14.287,Z -186.839,A -90.000,B 90.000,C 0.000} C_DIS
LIN {X -44.937,Y -14.287,Z -184.563,A -90.000,B 90.000,C 0.000} C_DIS
LIN {X -41.672,Y -14.287,Z -182.237,A -90.000,B 90.000,C 0.000} C_DIS
LIN {X -38.444,Y -14.287,Z -179.859,A -90.000,B 90.000,C 0.000} C_DIS
LIN {X -36.831,Y -14.287,Z -178.687,A -90.000,B 90.000,C 0.000} C_DIS
LIN {X -35.251,Y -14.287,Z -177.470,A -90.000,B 90.000,C 0.000} C_DIS
LIN {X -33.707,Y -14.287,Z -176.208,A -90.000,B 90.000,C 0.000} C_DIS
LIN {X -32.199,Y -14.287,Z -174.903,A -90.000,B 90.000,C 0.000} C_DIS
LIN {X -30.729,Y -14.287,Z -173.556,A -90.000,B 90.000,C 0.000} C_DIS
LIN {X -29.298,Y -14.287,Z -172.168,A -90.000,B 90.000,C 0.000} C_DIS
LIN {X -28.375,Y -14.287,Z -171.257,A -90.000,B 90.000,C 0.000} C_DIS
LIN {X -27.497,Y -14.287,Z -170.302,A -90.000,B 90.000,C 0.000} C_DIS
LIN {X -26.666,Y -14.287,Z -169.307,A -90.000,B 90.000,C 0.000} C_DIS
LIN {X -25.883,Y -14.287,Z -168.273,A -90.000,B 90.000,C 0.000} C_DIS
LIN {X -25.150,Y -14.287,Z -167.203,A -90.000,B 90.000,C 0.000} C_DIS
LIN {X -24.470,Y -14.287,Z -166.099,A -90.000,B 90.000,C 0.000} C_DIS
LIN {X -23.843,Y -14.287,Z -164.964,A -90.000,B 90.000,C 0.000} C_DIS
LIN {X -23.270,Y -14.287,Z -163.801,A -90.000,B 90.000,C 0.000} C_DIS
LIN {X -22.754,Y -14.287,Z -162.611,A -90.000,B 90.000,C 0.000} C_DIS
LIN {X -23.095,Y -14.287,Z -162.073,A -90.000,B 90.000,C 0.000} C_DIS
LIN {X -23.467,Y -14.287,Z -161.556,A -90.000,B 90.000,C 0.000} C_DIS
LIN {X -23.868,Y -14.287,Z -161.061,A -90.000,B 90.000,C 0.000} C_DIS
LIN {X -27.192,Y -14.287,Z -157.616,A -90.000,B 90.000,C 0.000} C_DIS
LIN {X -30.543,Y -14.287,Z -154.198,A -90.000,B 90.000,C 0.000} C_DIS
LIN {X -31.814,Y -14.287,Z -152.924,A -90.000,B 90.000,C 0.000} C_DIS
LIN {X -33.050,Y -14.287,Z -151.615,A -90.000,B 90.000,C 0.000} C_DIS
LIN {X -34.247,Y -14.287,Z -150.272,A -90.000,B 90.000,C 0.000} C_DIS
LIN {X -35.407,Y -14.287,Z -148.896,A -90.000,B 90.000,C 0.000} C_DIS
LIN {X -36.527,Y -14.287,Z -147.487,A -90.000,B 90.000,C 0.000} C_DIS
LIN {X -37.607,Y -14.287,Z -146.048,A -90.000,B 90.000,C 0.000} C_DIS
LIN {X -38.647,Y -14.287,Z -144.579,A -90.000,B 90.000,C 0.000} C_DIS
LIN {X -39.861,Y -14.287,Z -142.619,A -90.000,B 90.000,C 0.000} C_DIS
LIN {X -41.030,Y -14.287,Z -140.632,A -90.000,B 90.000,C 0.000} C_DIS
LIN {X -42.151,Y -14.287,Z -138.618,A -90.000,B 90.000,C 0.000} C_DIS
LIN {X -43.225,Y -14.287,Z -136.578,A -90.000,B 90.000,C 0.000} C_DIS
LIN {X -44.251,Y -14.287,Z -134.514,A -90.000,B 90.000,C 0.000} C_DIS
LIN {X -45.228,Y -14.287,Z -132.426,A -90.000,B 90.000,C 0.000} C_DIS
LIN {X -46.156,Y -14.287,Z -130.315,A -90.000,B 90.000,C 0.000} C_DIS
LIN {X -47.035,Y -14.287,Z -128.184,A -90.000,B 90.000,C 0.000} C_DIS
LIN {X -47.330,Y -14.287,Z -127.302,A -90.000,B 90.000,C 0.000} C_DIS
LIN {X -47.674,Y -14.287,Z -126.438,A -90.000,B 90.000,C 0.000} C_DIS
LIN {X -48.066,Y -14.287,Z -125.595,A -90.000,B 90.000,C 0.000} C_DIS
LIN {X -48.505,Y -14.287,Z -124.775,A -90.000,B 90.000,C 0.000} C_DIS
LIN {X -48.989,Y -14.287,Z -123.981,A -90.000,B 90.000,C 0.000} C_DIS
LIN {X -49.517,Y -14.287,Z -123.215,A -90.000,B 90.000,C 0.000} C_DIS
LIN {X -52.229,Y -14.287,Z -119.962,A -90.000,B 90.000,C 0.000} C_DIS
LIN {X -54.894,Y -14.287,Z -116.671,A -90.000,B 90.000,C 0.000} C_DIS
LIN {X -57.511,Y -14.287,Z -113.343,A -90.000,B 90.000,C 0.000} C_DIS
LIN {X -60.081,Y -14.287,Z -109.977,A -90.000,B 90.000,C 0.000} C_DIS
LIN {X -62.603,Y -14.287,Z -106.575,A -90.000,B 90.000,C 0.000} C_DIS
LIN {X -63.758,Y -14.287,Z -104.961,A -90.000,B 90.000,C 0.000} C_DIS
LIN {X -64.967,Y -14.287,Z -103.387,A -90.000,B 90.000,C 0.000} C_DIS
LIN {X -66.228,Y -14.287,Z -101.854,A -90.000,B 90.000,C 0.000} C_DIS
LIN {X -67.539,Y -14.287,Z -100.364,A -90.000,B 90.000,C 0.000} C_DIS
LIN {X -68.898,Y -14.287,Z -98.919,A -90.000,B 90.000,C 0.000} C_DIS
LIN {X -70.306,Y -14.287,Z -97.520,A -90.000,B 90.000,C 0.000} C_DIS
LIN {X -71.810,Y -14.287,Z -96.287,A -90.000,B 90.000,C 0.000} C_DIS
LIN {X -73.342,Y -14.287,Z -95.090,A -90.000,B 90.000,C 0.000} C_DIS
LIN {X -74.902,Y -14.287,Z -93.929,A -90.000,B 90.000,C 0.000} C_DIS
LIN {X -76.488,Y -14.287,Z -92.805,A -90.000,B 90.000,C 0.000} C_DIS
LIN {X -78.101,Y -14.287,Z -91.719,A -90.000,B 90.000,C 0.000} C_DIS
LIN {X -79.739,Y -14.287,Z -90.671,A -90.000,B 90.000,C 0.000} C_DIS
LIN {X -81.421,Y -14.287,Z -89.687,A -90.000,B 90.000,C 0.000} C_DIS
LIN {X -83.068,Y -14.287,Z -88.645,A -90.000,B 90.000,C 0.000} C_DIS
LIN {X -84.679,Y -14.287,Z -87.548,A -90.000,B 90.000,C 0.000} C_DIS
LIN {X -86.250,Y -14.287,Z -86.396,A -90.000,B 90.000,C 0.000} C_DIS
LIN {X -87.782,Y -14.287,Z -85.191,A -90.000,B 90.000,C 0.000} C_DIS
LIN {X -89.271,Y -14.287,Z -83.934,A -90.000,B 90.000,C 0.000} C_DIS
LIN {X -89.724,Y -14.287,Z -83.441,A -90.000,B 90.000,C 0.000} C_DIS
LIN {X -90.214,Y -14.287,Z -82.985,A -90.000,B 90.000,C 0.000} C_DIS
LIN {X -90.737,Y -14.287,Z -82.567,A -90.000,B 90.000,C 0.000} C_DIS
LIN {X -91.291,Y -14.287,Z -82.191,A -90.000,B 90.000,C 0.000} C_DIS
LIN {X -91.871,Y -14.287,Z -81.858,A -90.000,B 90.000,C 0.000} C_DIS
LIN {X -92.476,Y -14.287,Z -81.571,A -90.000,B 90.000,C 0.000} C_DIS
LIN {X -93.101,Y -14.287,Z -81.331,A -90.000,B 90.000,C 0.000} C_DIS
LIN {X -93.272,Y -14.287,Z -81.288,A -90.000,B 90.000,C 0.000} C_DIS
LIN {X -94.486,Y -14.287,Z -81.252,A -90.000,B 90.000,C 0.000} C_DIS
LIN {X -95.696,Y -14.287,Z -81.159,A -90.000,B 90.000,C 0.000} C_DIS
LIN {X -96.901,Y -14.287,Z -81.009,A -90.000,B 90.000,C 0.000} C_DIS
LIN {X -98.097,Y -14.287,Z -80.801,A -90.000,B 90.000,C 0.000} C_DIS
LIN {X -99.282,Y -14.287,Z -80.537,A -90.000,B 90.000,C 0.000} C_DIS
LIN {X -100.454,Y -14.287,Z -80.217,A -90.000,B 90.000,C 0.000} C_DIS
LIN {X -101.608,Y -14.287,Z -79.842,A -90.000,B 90.000,C 0.000} C_DIS
LIN {X -102.744,Y -14.287,Z -79.412,A -90.000,B 90.000,C 0.000} C_DIS
LIN {X -102.872,Y -14.287,Z -79.344,A -90.000,B 90.000,C 0.000} C_DIS
LIN {X -103.722,Y -14.287,Z -78.938,A -90.000,B 90.000,C 0.000} C_DIS
LIN {X -104.561,Y -14.287,Z -78.510,A -90.000,B 90.000,C 0.000} C_DIS
LIN {X -105.389,Y -14.287,Z -78.060,A -90.000,B 90.000,C 0.000} C_DIS
LIN {X -106.653,Y -14.287,Z -77.154,A -90.000,B 90.000,C 0.000} C_DIS
LIN {X -107.878,Y -14.287,Z -76.194,A -90.000,B 90.000,C 0.000} C_DIS
LIN {X -109.060,Y -14.287,Z -75.184,A -90.000,B 90.000,C 0.000} C_DIS
LIN {X -110.198,Y -14.287,Z -74.123,A -90.000,B 90.000,C 0.000} C_DIS
LIN {X -111.290,Y -14.287,Z -73.015,A -90.000,B 90.000,C 0.000} C_DIS
LIN {X -112.333,Y -14.287,Z -71.861,A -90.000,B 90.000,C 0.000} C_DIS
LIN {X -113.325,Y -14.287,Z -70.663,A -90.000,B 90.000,C 0.000} C_DIS
LIN {X -114.266,Y -14.287,Z -69.424,A -90.000,B 90.000,C 0.000} C_DIS
LIN {X -115.153,Y -14.287,Z -68.146,A -90.000,B 90.000,C 0.000} C_DIS
LIN {X -115.984,Y -14.287,Z -66.831,A -90.000,B 90.000,C 0.000} C_DIS
LIN {X -116.758,Y -14.287,Z -65.482,A -90.000,B 90.000,C 0.000} C_DIS
LIN {X -117.474,Y -14.287,Z -64.101,A -90.000,B 90.000,C 0.000} C_DIS
LIN {X -118.037,Y -14.287,Z -62.646,A -90.000,B 90.000,C 0.000} C_DIS
LIN {X -118.547,Y -14.287,Z -61.171,A -90.000,B 90.000,C 0.000} C_DIS
LIN {X -119.005,Y -14.287,Z -59.679,A -90.000,B 90.000,C 0.000} C_DIS
LIN {X -119.409,Y -14.287,Z -58.172,A -90.000,B 90.000,C 0.000} C_DIS
LIN {X -119.759,Y -14.287,Z -56.651,A -90.000,B 90.000,C 0.000} C_DIS
LIN {X -120.052,Y -14.287,Z -55.932,A -90.000,B 90.000,C 0.000} C_DIS
LIN {X -120.303,Y -14.287,Z -55.197,A -90.000,B 90.000,C 0.000} C_DIS
LIN {X -120.512,Y -14.287,Z -54.450,A -90.000,B 90.000,C 0.000} C_DIS
LIN {X -120.679,Y -14.287,Z -53.691,A -90.000,B 90.000,C 0.000} C_DIS
LIN {X -120.802,Y -14.287,Z -52.925,A -90.000,B 90.000,C 0.000} C_DIS
LIN {X -120.846,Y -14.287,Z -52.825,A -90.000,B 90.000,C 0.000} C_DIS
LIN {X -121.513,Y -14.287,Z -51.073,A -90.000,B 90.000,C 0.000} C_DIS
LIN {X -121.567,Y -14.287,Z -50.882,A -90.000,B 90.000,C 0.000} C_DIS
LIN {X -121.822,Y -14.287,Z -50.075,A -90.000,B 90.000,C 0.000} C_DIS
LIN {X -122.024,Y -14.287,Z -49.252,A -90.000,B 90.000,C 0.000} C_DIS
LIN {X -122.170,Y -14.287,Z -48.418,A -90.000,B 90.000,C 0.000} C_DIS
LIN {X -122.261,Y -14.287,Z -47.577,A -90.000,B 90.000,C 0.000} C_DIS
LIN {X -122.297,Y -14.287,Z -46.731,A -90.000,B 90.000,C 0.000} C_DIS
LIN {X -122.276,Y -14.287,Z -45.884,A -90.000,B 90.000,C 0.000} C_DIS
LIN {X -122.200,Y -14.287,Z -45.041,A -90.000,B 90.000,C 0.000} C_DIS
LIN {X -122.068,Y -14.287,Z -44.205,A -90.000,B 90.000,C 0.000} C_DIS
LIN {X -121.881,Y -14.287,Z -43.379,A -90.000,B 90.000,C 0.000} C_DIS
LIN {X -122.233,Y -14.287,Z -42.418,A -90.000,B 90.000,C 0.000} C_DIS
LIN {X -122.523,Y -14.287,Z -41.436,A -90.000,B 90.000,C 0.000} C_DIS
LIN {X -122.750,Y -14.287,Z -40.438,A -90.000,B 90.000,C 0.000} C_DIS
LIN {X -122.913,Y -14.287,Z -39.427,A -90.000,B 90.000,C 0.000} C_DIS
LIN {X -123.012,Y -14.287,Z -38.408,A -90.000,B 90.000,C 0.000} C_DIS
LIN {X -123.046,Y -14.287,Z -37.385,A -90.000,B 90.000,C 0.000} C_DIS
LIN {X -123.015,Y -14.287,Z -36.362,A -90.000,B 90.000,C 0.000} C_DIS
LIN {X -122.919,Y -14.287,Z -35.343,A -90.000,B 90.000,C 0.000} C_DIS
LIN {X -122.758,Y -14.287,Z -34.332,A -90.000,B 90.000,C 0.000} C_DIS
LIN {X -122.534,Y -14.287,Z -33.333,A -90.000,B 90.000,C 0.000} C_DIS
LIN {X -122.246,Y -14.287,Z -32.351,A -90.000,B 90.000,C 0.000} C_DIS
LIN {X -121.987,Y -14.287,Z -31.533,A -90.000,B 90.000,C 0.000} C_DIS
LIN {X -121.673,Y -14.287,Z -30.735,A -90.000,B 90.000,C 0.000} C_DIS
LIN {X -121.306,Y -14.287,Z -29.959,A -90.000,B 90.000,C 0.000} C_DIS
LIN {X -120.887,Y -14.287,Z -29.211,A -90.000,B 90.000,C 0.000} C_DIS
LIN {X -120.418,Y -14.287,Z -28.492,A -90.000,B 90.000,C 0.000} C_DIS
LIN {X -119.902,Y -14.287,Z -27.807,A -90.000,B 90.000,C 0.000} C_DIS
LIN {X -119.341,Y -14.287,Z -27.159,A -90.000,B 90.000,C 0.000} C_DIS
LIN {X -118.736,Y -14.287,Z -26.550,A -90.000,B 90.000,C 0.000} C_DIS
LIN {X -118.080,Y -14.287,Z -25.586,A -90.000,B 90.000,C 0.000} C_DIS
LIN {X -117.370,Y -14.287,Z -24.661,A -90.000,B 90.000,C 0.000} C_DIS
LIN {X -116.608,Y -14.287,Z -23.779,A -90.000,B 90.000,C 0.000} C_DIS
LIN {X -115.796,Y -14.287,Z -22.941,A -90.000,B 90.000,C 0.000} C_DIS
LIN {X -114.938,Y -14.287,Z -22.152,A -90.000,B 90.000,C 0.000} C_DIS
LIN {X -114.036,Y -14.287,Z -21.413,A -90.000,B 90.000,C 0.000} C_DIS
LIN {X -113.093,Y -14.287,Z -20.728,A -90.000,B 90.000,C 0.000} C_DIS
LIN {X -112.112,Y -14.287,Z -20.097,A -90.000,B 90.000,C 0.000} C_DIS
LIN {X -111.097,Y -14.287,Z -19.524,A -90.000,B 90.000,C 0.000} C_DIS
LIN {X -110.050,Y -14.287,Z -19.010,A -90.000,B 90.000,C 0.000} C_DIS
LIN {X -108.976,Y -14.287,Z -18.557,A -90.000,B 90.000,C 0.000} C_DIS
LIN {X -107.877,Y -14.287,Z -18.167,A -90.000,B 90.000,C 0.000} C_DIS
LIN {X -106.758,Y -14.287,Z -17.840,A -90.000,B 90.000,C 0.000} C_DIS
LIN {X -105.815,Y -14.287,Z -16.705,A -90.000,B 90.000,C 0.000} C_DIS
LIN {X -105.749,Y -14.287,Z -16.636,A -90.000,B 90.000,C 0.000} C_DIS
LIN {X -105.191,Y -14.287,Z -16.086,A -90.000,B 90.000,C 0.000} C_DIS
LIN {X -104.600,Y -14.287,Z -15.573,A -90.000,B 90.000,C 0.000} C_DIS
LIN {X -103.977,Y -14.287,Z -15.098,A -90.000,B 90.000,C 0.000} C_DIS
LIN {X -103.325,Y -14.287,Z -14.664,A -90.000,B 90.000,C 0.000} C_DIS
LIN {X -102.954,Y -14.287,Z -14.499,A -90.000,B 90.000,C 0.000} C_DIS
LIN {X -102.596,Y -14.287,Z -14.305,A -90.000,B 90.000,C 0.000} C_DIS
LIN {X -102.256,Y -14.287,Z -14.084,A -90.000,B 90.000,C 0.000} C_DIS
LIN {X -101.933,Y -14.287,Z -13.837,A -90.000,B 90.000,C 0.000} C_DIS
LIN {X -101.810,Y -14.287,Z -13.728,A -90.000,B 90.000,C 0.000} C_DIS
LIN {X -101.077,Y -14.287,Z -13.101,A -90.000,B 90.000,C 0.000} C_DIS
LIN {X -100.314,Y -14.287,Z -12.511,A -90.000,B 90.000,C 0.000} C_DIS
LIN {X -99.524,Y -14.287,Z -11.958,A -90.000,B 90.000,C 0.000} C_DIS
LIN {X -98.708,Y -14.287,Z -11.444,A -90.000,B 90.000,C 0.000} C_DIS
LIN {X -97.868,Y -14.287,Z -10.971,A -90.000,B 90.000,C 0.000} C_DIS
LIN {X -97.006,Y -14.287,Z -10.538,A -90.000,B 90.000,C 0.000} C_DIS
LIN {X -96.871,Y -14.287,Z -10.483,A -90.000,B 90.000,C 0.000} C_DIS
LIN {X -95.852,Y -14.287,Z -10.110,A -90.000,B 90.000,C 0.000} C_DIS
LIN {X -94.815,Y -14.287,Z -9.788,A -90.000,B 90.000,C 0.000} C_DIS
LIN {X -93.764,Y -14.287,Z -9.518,A -90.000,B 90.000,C 0.000} C_DIS
LIN {X -92.701,Y -14.287,Z -9.300,A -90.000,B 90.000,C 0.000} C_DIS
LIN {X -91.628,Y -14.287,Z -9.135,A -90.000,B 90.000,C 0.000} C_DIS
LIN {X -90.549,Y -14.287,Z -9.024,A -90.000,B 90.000,C 0.000} C_DIS
LIN {X -89.465,Y -14.287,Z -8.966,A -90.000,B 90.000,C 0.000} C_DIS
LIN {X -89.329,Y -14.287,Z -8.880,A -90.000,B 90.000,C 0.000} C_DIS
LIN {X -88.253,Y -14.287,Z -8.336,A -90.000,B 90.000,C 0.000} C_DIS
LIN {X -87.147,Y -14.287,Z -7.852,A -90.000,B 90.000,C 0.000} C_DIS
LIN {X -86.017,Y -14.287,Z -7.431,A -90.000,B 90.000,C 0.000} C_DIS
LIN {X -84.865,Y -14.287,Z -7.073,A -90.000,B 90.000,C 0.000} C_DIS
LIN {X -83.695,Y -14.287,Z -6.781,A -90.000,B 90.000,C 0.000} C_DIS
LIN {X -82.510,Y -14.287,Z -6.553,A -90.000,B 90.000,C 0.000} C_DIS
LIN {X -81.315,Y -14.287,Z -6.393,A -90.000,B 90.000,C 0.000} C_DIS
LIN {X -80.112,Y -14.287,Z -6.299,A -90.000,B 90.000,C 0.000} C_DIS
LIN {X -78.906,Y -14.287,Z -6.272,A -90.000,B 90.000,C 0.000} C_DIS
LIN {X -77.700,Y -14.287,Z -6.313,A -90.000,B 90.000,C 0.000} C_DIS
LIN {X -76.499,Y -14.287,Z -6.420,A -90.000,B 90.000,C 0.000} C_DIS
LIN {X -75.225,Y -14.287,Z -6.696,A -90.000,B 90.000,C 0.000} C_DIS
LIN {X -73.960,Y -14.287,Z -7.015,A -90.000,B 90.000,C 0.000} C_DIS
LIN {X -72.708,Y -14.287,Z -7.377,A -90.000,B 90.000,C 0.000} C_DIS
LIN {X -71.468,Y -14.287,Z -7.783,A -90.000,B 90.000,C 0.000} C_DIS
LIN {X -70.244,Y -14.287,Z -8.231,A -90.000,B 90.000,C 0.000} C_DIS
LIN {X -68.901,Y -14.287,Z -8.816,A -90.000,B 90.000,C 0.000} C_DIS
LIN {X -67.553,Y -14.287,Z -9.390,A -90.000,B 90.000,C 0.000} C_DIS
LIN {X -65.388,Y -14.287,Z -10.365,A -90.000,B 90.000,C 0.000} C_DIS
LIN {X -63.205,Y -14.287,Z -11.299,A -90.000,B 90.000,C 0.000} C_DIS
LIN {X -62.061,Y -14.287,Z -11.863,A -90.000,B 90.000,C 0.000} C_DIS
LIN {X -60.891,Y -14.287,Z -12.369,A -90.000,B 90.000,C 0.000} C_DIS
LIN {X -59.696,Y -14.287,Z -12.816,A -90.000,B 90.000,C 0.000} C_DIS
LIN {X -58.481,Y -14.287,Z -13.202,A -90.000,B 90.000,C 0.000} C_DIS
LIN {X -57.248,Y -14.287,Z -13.526,A -90.000,B 90.000,C 0.000} C_DIS
LIN {X -56.000,Y -14.287,Z -13.788,A -90.000,B 90.000,C 0.000} C_DIS
LIN {X -54.740,Y -14.287,Z -13.986,A -90.000,B 90.000,C 0.000} C_DIS
LIN {X -53.472,Y -14.287,Z -14.121,A -90.000,B 90.000,C 0.000} C_DIS
LIN {X -51.190,Y -14.287,Z -14.495,A -90.000,B 90.000,C 0.000} C_DIS
LIN {X -48.903,Y -14.287,Z -14.835,A -90.000,B 90.000,C 0.000} C_DIS
LIN {X -46.611,Y -14.287,Z -15.140,A -90.000,B 90.000,C 0.000} C_DIS
LIN {X -44.315,Y -14.287,Z -15.412,A -90.000,B 90.000,C 0.000} C_DIS
LIN {X -42.467,Y -14.287,Z -15.542,A -90.000,B 90.000,C 0.000} C_DIS
LIN {X -40.623,Y -14.287,Z -15.717,A -90.000,B 90.000,C 0.000} C_DIS
LIN {X -38.783,Y -14.287,Z -15.937,A -90.000,B 90.000,C 0.000} C_DIS
LIN {X -36.949,Y -14.287,Z -16.202,A -90.000,B 90.000,C 0.000} C_DIS
LIN {X -35.123,Y -14.287,Z -16.511,A -90.000,B 90.000,C 0.000} C_DIS
LIN {X -33.304,Y -14.287,Z -16.864,A -90.000,B 90.000,C 0.000} C_DIS
LIN {X -28.353,Y -14.287,Z -17.790,A -90.000,B 90.000,C 0.000} C_DIS
LIN {X -23.408,Y -14.287,Z -18.748,A -90.000,B 90.000,C 0.000} C_DIS
LIN {X -17.899,Y -14.287,Z -20.006,A -90.000,B 90.000,C 0.000} C_DIS
LIN {X -12.380,Y -14.287,Z -21.222,A -90.000,B 90.000,C 0.000} C_DIS
LIN {X -6.853,Y -14.287,Z -22.396,A -90.000,B 90.000,C 0.000} C_DIS
LIN {X -1.317,Y -14.287,Z -23.529,A -90.000,B 90.000,C 0.000} C_DIS
LIN {X 1.571,Y -14.287,Z -23.944,A -90.000,B 90.000,C 0.000} C_DIS
LIN {X 4.449,Y -14.287,Z -24.420,A -90.000,B 90.000,C 0.000} C_DIS
LIN {X 7.316,Y -14.287,Z -24.956,A -90.000,B 90.000,C 0.000} C_DIS
LIN {X 10.172,Y -14.287,Z -25.553,A -90.000,B 90.000,C 0.000} C_DIS
LIN {X 13.014,Y -14.287,Z -26.210,A -90.000,B 90.000,C 0.000} C_DIS
LIN {X 14.109,Y -14.287,Z -26.508,A -90.000,B 90.000,C 0.000} C_DIS
LIN {X 15.218,Y -14.287,Z -26.747,A -90.000,B 90.000,C 0.000} C_DIS
LIN {X 16.338,Y -14.287,Z -26.926,A -90.000,B 90.000,C 0.000} C_DIS
LIN {X 17.466,Y -14.287,Z -27.045,A -90.000,B 90.000,C 0.000} C_DIS
LIN {X 18.599,Y -14.287,Z -27.104,A -90.000,B 90.000,C 0.000} C_DIS
LIN {X 19.733,Y -14.287,Z -27.101,A -90.000,B 90.000,C 0.000} C_DIS
LIN {X 20.866,Y -14.287,Z -27.037,A -90.000,B 90.000,C 0.000} C_DIS
LIN {X 22.682,Y -14.287,Z -27.106,A -90.000,B 90.000,C 0.000} C_DIS
LIN {X 24.496,Y -14.287,Z -27.233,A -90.000,B 90.000,C 0.000} C_DIS
LIN {X 26.304,Y -14.287,Z -27.419,A -90.000,B 90.000,C 0.000} C_DIS
LIN {X 28.105,Y -14.287,Z -27.663,A -90.000,B 90.000,C 0.000} C_DIS
LIN {X 29.897,Y -14.287,Z -27.966,A -90.000,B 90.000,C 0.000} C_DIS
LIN {X 31.679,Y -14.287,Z -28.326,A -90.000,B 90.000,C 0.000} C_DIS
LIN {X 33.448,Y -14.287,Z -28.743,A -90.000,B 90.000,C 0.000} C_DIS
LIN {X 34.502,Y -14.287,Z -29.026,A -90.000,B 90.000,C 0.000} C_DIS
LIN {X 35.560,Y -14.287,Z -29.295,A -90.000,B 90.000,C 0.000} C_DIS
LIN {X 39.136,Y -14.287,Z -30.398,A -90.000,B 90.000,C 0.000} C_DIS
LIN {X 42.719,Y -14.287,Z -31.478,A -90.000,B 90.000,C 0.000} C_DIS
LIN {X 44.441,Y -14.287,Z -31.948,A -90.000,B 90.000,C 0.000} C_DIS
LIN {X 46.146,Y -14.287,Z -32.478,A -90.000,B 90.000,C 0.000} C_DIS
LIN {X 47.831,Y -14.287,Z -33.066,A -90.000,B 90.000,C 0.000} C_DIS
LIN {X 49.495,Y -14.287,Z -33.713,A -90.000,B 90.000,C 0.000} C_DIS
LIN {X 51.136,Y -14.287,Z -34.417,A -90.000,B 90.000,C 0.000} C_DIS
LIN {X 52.751,Y -14.287,Z -35.177,A -90.000,B 90.000,C 0.000} C_DIS
LIN {X 54.339,Y -14.287,Z -35.992,A -90.000,B 90.000,C 0.000} C_DIS
LIN {X 55.898,Y -14.287,Z -36.863,A -90.000,B 90.000,C 0.000} C_DIS
LIN {X 57.426,Y -14.287,Z -37.786,A -90.000,B 90.000,C 0.000} C_DIS
LIN {X 58.921,Y -14.287,Z -38.762,A -90.000,B 90.000,C 0.000} C_DIS
LIN {X 60.381,Y -14.287,Z -39.789,A -90.000,B 90.000,C 0.000} C_DIS
LIN {X 61.805,Y -14.287,Z -40.866,A -90.000,B 90.000,C 0.000} C_DIS
LIN {X 62.087,Y -14.287,Z -41.150,A -90.000,B 90.000,C 0.000} C_DIS
LIN {X 62.402,Y -14.287,Z -41.397,A -90.000,B 90.000,C 0.000} C_DIS
LIN {X 62.745,Y -14.287,Z -41.602,A -90.000,B 90.000,C 0.000} C_DIS
LIN {X 64.907,Y -14.287,Z -42.608,A -90.000,B 90.000,C 0.000} C_DIS
LIN {X 67.046,Y -14.287,Z -43.663,A -90.000,B 90.000,C 0.000} C_DIS
LIN {X 69.162,Y -14.287,Z -44.764,A -90.000,B 90.000,C 0.000} C_DIS
LIN {X 71.252,Y -14.287,Z -45.913,A -90.000,B 90.000,C 0.000} C_DIS
LIN {X 73.316,Y -14.287,Z -47.107,A -90.000,B 90.000,C 0.000} C_DIS
LIN {X 75.354,Y -14.287,Z -48.347,A -90.000,B 90.000,C 0.000} C_DIS
LIN {X 77.363,Y -14.287,Z -49.632,A -90.000,B 90.000,C 0.000} C_DIS
LIN {X 78.210,Y -14.287,Z -48.316,A -90.000,B 90.000,C 0.000} C_DIS
LIN {X 79.109,Y -14.287,Z -47.035,A -90.000,B 90.000,C 0.000} C_DIS
LIN {X 80.057,Y -14.287,Z -45.790,A -90.000,B 90.000,C 0.000} C_DIS
LIN {X 81.054,Y -14.287,Z -44.583,A -90.000,B 90.000,C 0.000} C_DIS
LIN {X 82.098,Y -14.287,Z -43.417,A -90.000,B 90.000,C 0.000} C_DIS
LIN {X 83.186,Y -14.287,Z -42.292,A -90.000,B 90.000,C 0.000} C_DIS
LIN {X 84.319,Y -14.287,Z -41.212,A -90.000,B 90.000,C 0.000} C_DIS
LIN {X 85.492,Y -14.287,Z -40.177,A -90.000,B 90.000,C 0.000} C_DIS
LIN {X 86.706,Y -14.287,Z -39.189,A -90.000,B 90.000,C 0.000} C_DIS
LIN {X 87.958,Y -14.287,Z -38.249,A -90.000,B 90.000,C 0.000} C_DIS
LIN {X 89.246,Y -14.287,Z -37.360,A -90.000,B 90.000,C 0.000} C_DIS
LIN {X 91.067,Y -14.287,Z -36.216,A -90.000,B 90.000,C 0.000} C_DIS
LIN {X 92.918,Y -14.287,Z -35.121,A -90.000,B 90.000,C 0.000} C_DIS
LIN {X 94.797,Y -14.287,Z -34.076,A -90.000,B 90.000,C 0.000} C_DIS
LIN {X 96.704,Y -14.287,Z -33.081,A -90.000,B 90.000,C 0.000} C_DIS
LIN {X 98.636,Y -14.287,Z -32.137,A -90.000,B 90.000,C 0.000} C_DIS
LIN {X 100.592,Y -14.287,Z -31.245,A -90.000,B 90.000,C 0.000} C_DIS
LIN {X 102.572,Y -14.287,Z -30.405,A -90.000,B 90.000,C 0.000} C_DIS
LIN {X 104.573,Y -14.287,Z -29.618,A -90.000,B 90.000,C 0.000} C_DIS
LIN {X 105.490,Y -14.287,Z -29.228,A -90.000,B 90.000,C 0.000} C_DIS
LIN {X 106.432,Y -14.287,Z -28.905,A -90.000,B 90.000,C 0.000} C_DIS
LIN {X 107.394,Y -14.287,Z -28.649,A -90.000,B 90.000,C 0.000} C_DIS
LIN {X 108.372,Y -14.287,Z -28.462,A -90.000,B 90.000,C 0.000} C_DIS
LIN {X 109.361,Y -14.287,Z -28.344,A -90.000,B 90.000,C 0.000} C_DIS
LIN {X 110.356,Y -14.287,Z -28.297,A -90.000,B 90.000,C 0.000} C_DIS
LIN {X 111.352,Y -14.287,Z -28.321,A -90.000,B 90.000,C 0.000} C_DIS
LIN {X 112.343,Y -14.287,Z -28.416,A -90.000,B 90.000,C 0.000} C_DIS
LIN {X 113.326,Y -14.287,Z -28.580,A -90.000,B 90.000,C 0.000} C_DIS
LIN {X 114.294,Y -14.287,Z -28.814,A -90.000,B 90.000,C 0.000} C_DIS
LIN {X 115.243,Y -14.287,Z -29.116,A -90.000,B 90.000,C 0.000} C_DIS
LIN {X 116.168,Y -14.287,Z -29.484,A -90.000,B 90.000,C 0.000} C_DIS
LIN {X 117.065,Y -14.287,Z -29.917,A -90.000,B 90.000,C 0.000} C_DIS
LIN {X 117.929,Y -14.287,Z -30.413,A -90.000,B 90.000,C 0.000} C_DIS
LIN {X 118.756,Y -14.287,Z -30.969,A -90.000,B 90.000,C 0.000} C_DIS
LIN {X 119.541,Y -14.287,Z -31.582,A -90.000,B 90.000,C 0.000} C_DIS
LIN {X 120.281,Y -14.287,Z -32.248,A -90.000,B 90.000,C 0.000} C_DIS
LIN {X 120.415,Y -14.287,Z -32.376,A -90.000,B 90.000,C 0.000} C_DIS
LIN {X 121.045,Y -14.287,Z -33.072,A -90.000,B 90.000,C 0.000} C_DIS
LIN {X 121.662,Y -14.287,Z -33.780,A -90.000,B 90.000,C 0.000} C_DIS
LIN {X 122.196,Y -14.287,Z -34.612,A -90.000,B 90.000,C 0.000} C_DIS
LIN {X 122.676,Y -14.287,Z -35.476,A -90.000,B 90.000,C 0.000} C_DIS
LIN {X 123.102,Y -14.287,Z -36.368,A -90.000,B 90.000,C 0.000} C_DIS
LIN {X 123.470,Y -14.287,Z -37.286,A -90.000,B 90.000,C 0.000} C_DIS
LIN {X 123.781,Y -14.287,Z -38.224,A -90.000,B 90.000,C 0.000} C_DIS
LIN {X 124.032,Y -14.287,Z -39.180,A -90.000,B 90.000,C 0.000} C_DIS
LIN {X 124.222,Y -14.287,Z -40.150,A -90.000,B 90.000,C 0.000} C_DIS
LIN {X 124.352,Y -14.287,Z -41.130,A -90.000,B 90.000,C 0.000} C_DIS
LIN {X 124.419,Y -14.287,Z -42.117,A -90.000,B 90.000,C 0.000} C_DIS
LIN {X 124.425,Y -14.287,Z -43.105,A -90.000,B 90.000,C 0.000} C_DIS
LIN {X 124.369,Y -14.287,Z -44.092,A -90.000,B 90.000,C 0.000} C_DIS
LIN {X 124.170,Y -14.287,Z -45.366,A -90.000,B 90.000,C 0.000} C_DIS
LIN {X 123.911,Y -14.287,Z -46.630,A -90.000,B 90.000,C 0.000} C_DIS
LIN {X 123.595,Y -14.287,Z -47.880,A -90.000,B 90.000,C 0.000} C_DIS
LIN {X 123.220,Y -14.287,Z -49.114,A -90.000,B 90.000,C 0.000} C_DIS
LIN {X 122.789,Y -14.287,Z -50.330,A -90.000,B 90.000,C 0.000} C_DIS
LIN {X 122.302,Y -14.287,Z -51.524,A -90.000,B 90.000,C 0.000} C_DIS
LIN {X 121.760,Y -14.287,Z -52.694,A -90.000,B 90.000,C 0.000} C_DIS
LIN {X 121.061,Y -14.287,Z -53.939,A -90.000,B 90.000,C 0.000} C_DIS
LIN {X 120.409,Y -14.287,Z -55.208,A -90.000,B 90.000,C 0.000} C_DIS
LIN {X 119.804,Y -14.287,Z -56.501,A -90.000,B 90.000,C 0.000} C_DIS
LIN {X 119.247,Y -14.287,Z -57.815,A -90.000,B 90.000,C 0.000} C_DIS
LIN {X 118.739,Y -14.287,Z -59.149,A -90.000,B 90.000,C 0.000} C_DIS
LIN {X 118.281,Y -14.287,Z -60.500,A -90.000,B 90.000,C 0.000} C_DIS
LIN {X 117.872,Y -14.287,Z -61.868,A -90.000,B 90.000,C 0.000} C_DIS
LIN {X 117.373,Y -14.287,Z -63.949,A -90.000,B 90.000,C 0.000} C_DIS
LIN {X 116.813,Y -14.287,Z -66.015,A -90.000,B 90.000,C 0.000} C_DIS
LIN {X 116.194,Y -14.287,Z -68.064,A -90.000,B 90.000,C 0.000} C_DIS
LIN {X 115.517,Y -14.287,Z -70.095,A -90.000,B 90.000,C 0.000} C_DIS
LIN {X 114.780,Y -14.287,Z -72.104,A -90.000,B 90.000,C 0.000} C_DIS
LIN {X 113.986,Y -14.287,Z -74.092,A -90.000,B 90.000,C 0.000} C_DIS
LIN {X 113.134,Y -14.287,Z -76.056,A -90.000,B 90.000,C 0.000} C_DIS
LIN {X 112.226,Y -14.287,Z -77.994,A -90.000,B 90.000,C 0.000} C_DIS
LIN {X 111.262,Y -14.287,Z -79.905,A -90.000,B 90.000,C 0.000} C_DIS
LIN {X 110.244,Y -14.287,Z -81.787,A -90.000,B 90.000,C 0.000} C_DIS
LIN {X 109.171,Y -14.287,Z -83.640,A -90.000,B 90.000,C 0.000} C_DIS
LIN {X 108.045,Y -14.287,Z -85.460,A -90.000,B 90.000,C 0.000} C_DIS
LIN {X 108.619,Y -14.287,Z -86.520,A -90.000,B 90.000,C 0.000} C_DIS
LIN {X 109.147,Y -14.287,Z -87.603,A -90.000,B 90.000,C 0.000} C_DIS
LIN {X 109.630,Y -14.287,Z -88.708,A -90.000,B 90.000,C 0.000} C_DIS
LIN {X 110.065,Y -14.287,Z -89.832,A -90.000,B 90.000,C 0.000} C_DIS
LIN {X 110.452,Y -14.287,Z -90.973,A -90.000,B 90.000,C 0.000} C_DIS
LIN {X 111.322,Y -14.287,Z -94.510,A -90.000,B 90.000,C 0.000} C_DIS
LIN {X 112.124,Y -14.287,Z -98.062,A -90.000,B 90.000,C 0.000} C_DIS
LIN {X 112.857,Y -14.287,Z -101.630,A -90.000,B 90.000,C 0.000} C_DIS
LIN {X 113.520,Y -14.287,Z -105.211,A -90.000,B 90.000,C 0.000} C_DIS
LIN {X 114.115,Y -14.287,Z -108.804,A -90.000,B 90.000,C 0.000} C_DIS
LIN {X 114.639,Y -14.287,Z -112.409,A -90.000,B 90.000,C 0.000} C_DIS
LIN {X 115.094,Y -14.287,Z -116.022,A -90.000,B 90.000,C 0.000} C_DIS
LIN {X 115.478,Y -14.287,Z -119.644,A -90.000,B 90.000,C 0.000} C_DIS
LIN {X 115.793,Y -14.287,Z -123.272,A -90.000,B 90.000,C 0.000} C_DIS
LIN {X 116.037,Y -14.287,Z -126.906,A -90.000,B 90.000,C 0.000} C_DIS
LIN {X 116.210,Y -14.287,Z -130.544,A -90.000,B 90.000,C 0.000} C_DIS
LIN {X 116.314,Y -14.287,Z -134.185,A -90.000,B 90.000,C 0.000} C_DIS
LIN {X 116.346,Y -14.287,Z -137.827,A -90.000,B 90.000,C 0.000} C_DIS
LIN {X 116.309,Y -14.287,Z -141.469,A -90.000,B 90.000,C 0.000} C_DIS
LIN {X 116.200,Y -14.287,Z -145.109,A -90.000,B 90.000,C 0.000} C_DIS
LIN {X 116.022,Y -14.287,Z -148.747,A -90.000,B 90.000,C 0.000} C_DIS
LIN {X 115.567,Y -14.287,Z -154.512,A -90.000,B 90.000,C 0.000} C_DIS
LIN {X 115.044,Y -14.287,Z -160.270,A -90.000,B 90.000,C 0.000} C_DIS
LIN {X 114.454,Y -14.287,Z -166.023,A -90.000,B 90.000,C 0.000} C_DIS
LIN {X 113.796,Y -14.287,Z -171.768,A -90.000,B 90.000,C 0.000} C_DIS
LIN {X 113.070,Y -14.287,Z -177.505,A -90.000,B 90.000,C 0.000} C_DIS
LIN {X 112.277,Y -14.287,Z -183.233,A -90.000,B 90.000,C 0.000} C_DIS
LIN {X 111.417,Y -14.287,Z -188.951,A -90.000,B 90.000,C 0.000} C_DIS
LIN {X 110.489,Y -14.287,Z -194.658,A -90.000,B 90.000,C 0.000} C_DIS
LIN {X 109.495,Y -14.287,Z -200.355,A -90.000,B 90.000,C 0.000} C_DIS
LIN {X 108.433,Y -14.287,Z -206.039,A -90.000,B 90.000,C 0.000} C_DIS
LIN {X 107.652,Y -14.287,Z -210.273,A -90.000,B 90.000,C 0.000} C_DIS
LIN {X 106.800,Y -14.287,Z -214.493,A -90.000,B 90.000,C 0.000} C_DIS
LIN {X 105.879,Y -14.287,Z -218.699,A -90.000,B 90.000,C 0.000} C_DIS
LIN {X 104.889,Y -14.287,Z -222.889,A -90.000,B 90.000,C 0.000} C_DIS
LIN {X 103.830,Y -14.287,Z -227.061,A -90.000,B 90.000,C 0.000} C_DIS
LIN {X 102.701,Y -14.287,Z -231.216,A -90.000,B 90.000,C 0.000} C_DIS
LIN {X 101.504,Y -14.287,Z -235.352,A -90.000,B 90.000,C 0.000} C_DIS
LIN {X 100.239,Y -14.287,Z -239.467,A -90.000,B 90.000,C 0.000} C_DIS
LIN {X 98.907,Y -14.287,Z -243.561,A -90.000,B 90.000,C 0.000} C_DIS
LIN {X 145.015,Y -14.287,Z -243.561,A -90.000,B 90.000,C 0.000} C_DIS
LIN {X 145.015,Y -26.788,Z -243.561,A -90.000,B 90.000,C 0.000} C_DIS
LIN {X 145.015,Y -39.288,Z -243.561,A -90.000,B 90.000,C 0.000} C_DIS
LIN {X 145.015,Y -57.084,Z -243.561,A -90.000,B 90.000,C 0.000} C_DIS
LIN {X -144.015,Y -57.084,Z -242.561,A -90.000,B 90.000,C 0.000} C_DIS
LIN {X -144.015,Y -32.144,Z -242.561,A -90.000,B 90.000,C 0.000} C_DIS
LIN {X -144.015,Y -19.644,Z -242.561,A -90.000,B 90.000,C 0.000} C_DIS
LIN {X -144.015,Y -7.144,Z -242.561,A -90.000,B 90.000,C 0.000} C_DIS
LIN {X -141.117,Y -7.144,Z -242.561,A -90.000,B 90.000,C 0.000} C_DIS
LIN {X -140.672,Y -7.144,Z -241.914,A -90.000,B 90.000,C 0.000} C_DIS
LIN {X -140.186,Y -7.144,Z -241.297,A -90.000,B 90.000,C 0.000} C_DIS
LIN {X -139.661,Y -7.144,Z -240.713,A -90.000,B 90.000,C 0.000} C_DIS
LIN {X -139.098,Y -7.144,Z -240.165,A -90.000,B 90.000,C 0.000} C_DIS
LIN {X -138.501,Y -7.144,Z -239.655,A -90.000,B 90.000,C 0.000} C_DIS
LIN {X -136.227,Y -7.144,Z -238.069,A -90.000,B 90.000,C 0.000} C_DIS
LIN {X -133.928,Y -7.144,Z -236.521,A -90.000,B 90.000,C 0.000} C_DIS
LIN {X -131.603,Y -7.144,Z -235.012,A -90.000,B 90.000,C 0.000} C_DIS
LIN {X -144.015,Y -7.144,Z -235.012,A -90.000,B 90.000,C 0.000} C_DIS
LIN {X -144.015,Y -7.144,Z -227.464,A -90.000,B 90.000,C 0.000} C_DIS
LIN {X -120.059,Y -7.144,Z -227.464,A -90.000,B 90.000,C 0.000} C_DIS
LIN {X -115.823,Y -7.144,Z -224.683,A -90.000,B 90.000,C 0.000} C_DIS
LIN {X -112.164,Y -7.144,Z -222.287,A -90.000,B 90.000,C 0.000} C_DIS
LIN {X -108.489,Y -7.144,Z -219.915,A -90.000,B 90.000,C 0.000} C_DIS
LIN {X -144.015,Y -7.144,Z -219.915,A -90.000,B 90.000,C 0.000} C_DIS
LIN {X -144.015,Y -7.144,Z -212.366,A -90.000,B 90.000,C 0.000} C_DIS
LIN {X -96.426,Y -7.144,Z -212.366,A -90.000,B 90.000,C 0.000} C_DIS
LIN {X -92.221,Y -7.144,Z -209.818,A -90.000,B 90.000,C 0.000} C_DIS
LIN {X -87.998,Y -7.144,Z -207.302,A -90.000,B 90.000,C 0.000} C_DIS
LIN {X -83.756,Y -7.144,Z -204.817,A -90.000,B 90.000,C 0.000} C_DIS
LIN {X -144.015,Y -7.144,Z -204.817,A -90.000,B 90.000,C 0.000} C_DIS
LIN {X -144.015,Y -7.144,Z -197.269,A -90.000,B 90.000,C 0.000} C_DIS
LIN {X -70.385,Y -7.144,Z -197.269,A -90.000,B 90.000,C 0.000} C_DIS
LIN {X -66.002,Y -7.144,Z -194.795,A -90.000,B 90.000,C 0.000} C_DIS
LIN {X -61.642,Y -7.144,Z -192.279,A -90.000,B 90.000,C 0.000} C_DIS
LIN {X -57.308,Y -7.144,Z -189.720,A -90.000,B 90.000,C 0.000} C_DIS
LIN {X -144.015,Y -7.144,Z -189.720,A -90.000,B 90.000,C 0.000} C_DIS
LIN {X -144.015,Y -7.144,Z -182.171,A -90.000,B 90.000,C 0.000} C_DIS
LIN {X -45.342,Y -7.144,Z -182.171,A -90.000,B 90.000,C 0.000} C_DIS
LIN {X -43.278,Y -7.144,Z -180.726,A -90.000,B 90.000,C 0.000} C_DIS
LIN {X -41.237,Y -7.144,Z -179.248,A -90.000,B 90.000,C 0.000} C_DIS
LIN {X -39.220,Y -7.144,Z -177.738,A -90.000,B 90.000,C 0.000} C_DIS
LIN {X -37.227,Y -7.144,Z -176.196,A -90.000,B 90.000,C 0.000} C_DIS
LIN {X -35.259,Y -7.144,Z -174.622,A -90.000,B 90.000,C 0.000} C_DIS
LIN {X -144.015,Y -7.144,Z -174.622,A -90.000,B 90.000,C 0.000} C_DIS
LIN {X -144.015,Y -7.144,Z -167.073,A -90.000,B 90.000,C 0.000} C_DIS
LIN {X -28.079,Y -7.144,Z -167.073,A -90.000,B 90.000,C 0.000} C_DIS
LIN {X -27.537,Y -7.144,Z -166.179,A -90.000,B 90.000,C 0.000} C_DIS
LIN {X -27.031,Y -7.144,Z -165.264,A -90.000,B 90.000,C 0.000} C_DIS
LIN {X -26.564,Y -7.144,Z -164.328,A -90.000,B 90.000,C 0.000} C_DIS
LIN {X -26.134,Y -7.144,Z -163.375,A -90.000,B 90.000,C 0.000} C_DIS
LIN {X -25.744,Y -7.144,Z -162.405,A -90.000,B 90.000,C 0.000} C_DIS
LIN {X -26.481,Y -7.144,Z -161.426,A -90.000,B 90.000,C 0.000} C_DIS
LIN {X -27.242,Y -7.144,Z -160.466,A -90.000,B 90.000,C 0.000} C_DIS
LIN {X -28.027,Y -7.144,Z -159.525,A -90.000,B 90.000,C 0.000} C_DIS
LIN {X -144.015,Y -7.144,Z -159.525,A -90.000,B 90.000,C 0.000} C_DIS
LIN {X -144.015,Y -7.144,Z -151.976,A -90.000,B 90.000,C 0.000} C_DIS
LIN {X -35.060,Y -7.144,Z -151.976,A -90.000,B 90.000,C 0.000} C_DIS
LIN {X -36.113,Y -7.144,Z -150.710,A -90.000,B 90.000,C 0.000} C_DIS
LIN {X -37.139,Y -7.144,Z -149.421,A -90.000,B 90.000,C 0.000} C_DIS
LIN {X -38.136,Y -7.144,Z -148.110,A -90.000,B 90.000,C 0.000} C_DIS
LIN {X -39.104,Y -7.144,Z -146.778,A -90.000,B 90.000,C 0.000} C_DIS
LIN {X -39.872,Y -7.144,Z -145.608,A -90.000,B 90.000,C 0.000} C_DIS
LIN {X -40.621,Y -7.144,Z -144.427,A -90.000,B 90.000,C 0.000} C_DIS
LIN {X -144.015,Y -7.144,Z -144.427,A -90.000,B 90.000,C 0.000} C_DIS
LIN {X -144.015,Y -7.144,Z -136.878,A -90.000,B 90.000,C 0.000} C_DIS
LIN {X -44.841,Y -7.144,Z -136.878,A -90.000,B 90.000,C 0.000} C_DIS
LIN {X -45.661,Y -7.144,Z -135.188,A -90.000,B 90.000,C 0.000} C_DIS
LIN {X -46.445,Y -7.144,Z -133.482,A -90.000,B 90.000,C 0.000} C_DIS
LIN {X -47.194,Y -7.144,Z -131.760,A -90.000,B 90.000,C 0.000} C_DIS
LIN {X -47.668,Y -7.144,Z -130.539,A -90.000,B 90.000,C 0.000} C_DIS
LIN {X -48.168,Y -7.144,Z -129.329,A -90.000,B 90.000,C 0.000} C_DIS
LIN {X -144.015,Y -7.144,Z -129.329,A -90.000,B 90.000,C 0.000} C_DIS
LIN {X -144.015,Y -7.144,Z -121.781,A -90.000,B 90.000,C 0.000} C_DIS
LIN {X -52.583,Y -7.144,Z -121.781,A -90.000,B 90.000,C 0.000} C_DIS
LIN {X -53.297,Y -7.144,Z -120.877,A -90.000,B 90.000,C 0.000} C_DIS
LIN {X -54.029,Y -7.144,Z -119.988,A -90.000,B 90.000,C 0.000} C_DIS
LIN {X -55.542,Y -7.144,Z -118.054,A -90.000,B 90.000,C 0.000} C_DIS
LIN {X -57.073,Y -7.144,Z -116.136,A -90.000,B 90.000,C 0.000} C_DIS
LIN {X -58.623,Y -7.144,Z -114.232,A -90.000,B 90.000,C 0.000} C_DIS
LIN {X -144.015,Y -7.144,Z -114.232,A -90.000,B 90.000,C 0.000} C_DIS
LIN {X -144.015,Y -7.144,Z -106.683,A -90.000,B 90.000,C 0.000} C_DIS
LIN {X -65.086,Y -7.144,Z -106.683,A -90.000,B 90.000,C 0.000} C_DIS
LIN {X -65.176,Y -7.144,Z -106.583,A -90.000,B 90.000,C 0.000} C_DIS
LIN {X -66.442,Y -7.144,Z -105.248,A -90.000,B 90.000,C 0.000} C_DIS
LIN {X -67.746,Y -7.144,Z -103.949,A -90.000,B 90.000,C 0.000} C_DIS
LIN {X -69.085,Y -7.144,Z -102.687,A -90.000,B 90.000,C 0.000} C_DIS
LIN {X -70.459,Y -7.144,Z -101.464,A -90.000,B 90.000,C 0.000} C_DIS
LIN {X -71.868,Y -7.144,Z -100.279,A -90.000,B 90.000,C 0.000} C_DIS
LIN {X -73.308,Y -7.144,Z -99.134,A -90.000,B 90.000,C 0.000} C_DIS
LIN {X -144.015,Y -7.144,Z -99.134,A -90.000,B 90.000,C 0.000} C_DIS
LIN {X -144.015,Y -7.144,Z -91.586,A -90.000,B 90.000,C 0.000} C_DIS
LIN {X -84.422,Y -7.144,Z -91.586,A -90.000,B 90.000,C 0.000} C_DIS
LIN {X -86.679,Y -7.144,Z -89.913,A -90.000,B 90.000,C 0.000} C_DIS
LIN {X -88.944,Y -7.144,Z -88.252,A -90.000,B 90.000,C 0.000} C_DIS
LIN {X -90.652,Y -7.144,Z -87.093,A -90.000,B 90.000,C 0.000} C_DIS
LIN {X -92.347,Y -7.144,Z -85.917,A -90.000,B 90.000,C 0.000} C_DIS
LIN {X -93.628,Y -7.144,Z -85.987,A -90.000,B 90.000,C 0.000} C_DIS
LIN {X -94.910,Y -7.144,Z -85.994,A -90.000,B 90.000,C 0.000} C_DIS
LIN {X -96.192,Y -7.144,Z -85.938,A -90.000,B 90.000,C 0.000} C_DIS
LIN {X -97.469,Y -7.144,Z -85.819,A -90.000,B 90.000,C 0.000} C_DIS
LIN {X -98.739,Y -7.144,Z -85.637,A -90.000,B 90.000,C 0.000} C_DIS
LIN {X -99.998,Y -7.144,Z -85.393,A -90.000,B 90.000,C 0.000} C_DIS
LIN {X -101.243,Y -7.144,Z -85.087,A -90.000,B 90.000,C 0.000} C_DIS
LIN {X -102.472,Y -7.144,Z -84.720,A -90.000,B 90.000,C 0.000} C_DIS
LIN {X -103.682,Y -7.144,Z -84.293,A -90.000,B 90.000,C 0.000} C_DIS
LIN {X -104.243,Y -7.144,Z -84.037,A -90.000,B 90.000,C 0.000} C_DIS
LIN {X -144.015,Y -7.144,Z -84.037,A -90.000,B 90.000,C 0.000} C_DIS
LIN {X -144.015,Y -7.144,Z -76.488,A -90.000,B 90.000,C 0.000} C_DIS
LIN {X -114.751,Y -7.144,Z -76.488,A -90.000,B 90.000,C 0.000} C_DIS
LIN {X -115.666,Y -7.144,Z -75.490,A -90.000,B 90.000,C 0.000} C_DIS
LIN {X -116.541,Y -7.144,Z -74.458,A -90.000,B 90.000,C 0.000} C_DIS
LIN {X -117.375,Y -7.144,Z -73.392,A -90.000,B 90.000,C 0.000} C_DIS
LIN {X -118.168,Y -7.144,Z -72.295,A -90.000,B 90.000,C 0.000} C_DIS
LIN {X -118.783,Y -7.144,Z -71.191,A -90.000,B 90.000,C 0.000} C_DIS
LIN {X -119.369,Y -7.144,Z -70.072,A -90.000,B 90.000,C 0.000} C_DIS
LIN {X -119.928,Y -7.144,Z -68.939,A -90.000,B 90.000,C 0.000} C_DIS
LIN {X -144.015,Y -7.144,Z -68.939,A -90.000,B 90.000,C 0.000} C_DIS
LIN {X -144.015,Y -7.144,Z -61.390,A -90.000,B 90.000,C 0.000} C_DIS
LIN {X -122.860,Y -7.144,Z -61.390,A -90.000,B 90.000,C 0.000} C_DIS
LIN {X -123.592,Y -7.144,Z -59.258,A -90.000,B 90.000,C 0.000} C_DIS
LIN {X -124.057,Y -7.144,Z -58.204,A -90.000,B 90.000,C 0.000} C_DIS
LIN {X -124.485,Y -7.144,Z -57.134,A -90.000,B 90.000,C 0.000} C_DIS
LIN {X -124.873,Y -7.144,Z -56.050,A -90.000,B 90.000,C 0.000} C_DIS
LIN {X -125.222,Y -7.144,Z -54.952,A -90.000,B 90.000,C 0.000} C_DIS
LIN {X -125.532,Y -7.144,Z -53.842,A -90.000,B 90.000,C 0.000} C_DIS
LIN {X -144.015,Y -7.144,Z -53.842,A -90.000,B 90.000,C 0.000} C_DIS
LIN {X -144.015,Y -7.144,Z -46.293,A -90.000,B 90.000,C 0.000} C_DIS
LIN {X -126.157,Y -7.144,Z -46.293,A -90.000,B 90.000,C 0.000} C_DIS
LIN {X -126.148,Y -7.144,Z -46.236,A -90.000,B 90.000,C 0.000} C_DIS
LIN {X -126.554,Y -7.144,Z -44.508,A -90.000,B 90.000,C 0.000} C_DIS
LIN {X -126.734,Y -7.144,Z -43.558,A -90.000,B 90.000,C 0.000} C_DIS
LIN {X -126.850,Y -7.144,Z -42.598,A -90.000,B 90.000,C 0.000} C_DIS
LIN {X -126.903,Y -7.144,Z -41.632,A -90.000,B 90.000,C 0.000} C_DIS
LIN {X -126.890,Y -7.144,Z -40.665,A -90.000,B 90.000,C 0.000} C_DIS
LIN {X -126.814,Y -7.144,Z -39.701,A -90.000,B 90.000,C 0.000} C_DIS
LIN {X -126.674,Y -7.144,Z -38.744,A -90.000,B 90.000,C 0.000} C_DIS
LIN {X -144.015,Y -7.144,Z -38.744,A -90.000,B 90.000,C 0.000} C_DIS
LIN {X -144.015,Y -7.144,Z -31.195,A -90.000,B 90.000,C 0.000} C_DIS
LIN {X -126.091,Y -7.144,Z -31.195,A -90.000,B 90.000,C 0.000} C_DIS
LIN {X -125.875,Y -7.144,Z -30.176,A -90.000,B 90.000,C 0.000} C_DIS
LIN {X -125.598,Y -7.144,Z -29.172,A -90.000,B 90.000,C 0.000} C_DIS
LIN {X -125.262,Y -7.144,Z -28.185,A -90.000,B 90.000,C 0.000} C_DIS
LIN {X -124.869,Y -7.144,Z -27.221,A -90.000,B 90.000,C 0.000} C_DIS
LIN {X -124.418,Y -7.144,Z -26.281,A -90.000,B 90.000,C 0.000} C_DIS
LIN {X -123.913,Y -7.144,Z -25.370,A -90.000,B 90.000,C 0.000} C_DIS
LIN {X -123.354,Y -7.144,Z -24.491,A -90.000,B 90.000,C 0.000} C_DIS
LIN {X -122.745,Y -7.144,Z -23.646,A -90.000,B 90.000,C 0.000} C_DIS
LIN {X -144.015,Y -7.144,Z -23.646,A -90.000,B 90.000,C 0.000} C_DIS
LIN {X -144.015,Y -7.144,Z -16.098,A -90.000,B 90.000,C 0.000} C_DIS
LIN {X -116.332,Y -7.144,Z -16.098,A -90.000,B 90.000,C 0.000} C_DIS
LIN {X -115.380,Y -7.144,Z -15.441,A -90.000,B 90.000,C 0.000} C_DIS
LIN {X -114.396,Y -7.144,Z -14.834,A -90.000,B 90.000,C 0.000} C_DIS
LIN {X -113.382,Y -7.144,Z -14.278,A -90.000,B 90.000,C 0.000} C_DIS
LIN {X -112.340,Y -7.144,Z -13.776,A -90.000,B 90.000,C 0.000} C_DIS
LIN {X -111.273,Y -7.144,Z -13.329,A -90.000,B 90.000,C 0.000} C_DIS
LIN {X -110.185,Y -7.144,Z -12.937,A -90.000,B 90.000,C 0.000} C_DIS
LIN {X -109.078,Y -7.144,Z -12.602,A -90.000,B 90.000,C 0.000} C_DIS
LIN {X -107.955,Y -7.144,Z -12.326,A -90.000,B 90.000,C 0.000} C_DIS
LIN {X -106.820,Y -7.144,Z -12.107,A -90.000,B 90.000,C 0.000} C_DIS
LIN {X -105.674,Y -7.144,Z -11.948,A -90.000,B 90.000,C 0.000} C_DIS
LIN {X -104.753,Y -7.144,Z -11.261,A -90.000,B 90.000,C 0.000} C_DIS
LIN {X -103.513,Y -7.144,Z -10.536,A -90.000,B 90.000,C 0.000} C_DIS
LIN {X -102.256,Y -7.144,Z -9.842,A -90.000,B 90.000,C 0.000} C_DIS
LIN {X -100.982,Y -7.144,Z -9.180,A -90.000,B 90.000,C 0.000} C_DIS
LIN {X -99.692,Y -7.144,Z -8.549,A -90.000,B 90.000,C 0.000} C_DIS
LIN {X -144.015,Y -7.144,Z -8.549,A -90.000,B 90.000,C 0.000} C_DIS
LIN {X -144.015,Y -7.144,Z -1.000,A -90.000,B 90.000,C 0.000} C_DIS
LIN {X 144.015,Y -7.144,Z -1.000,A -90.000,B 90.000,C 0.000} C_DIS
LIN {X 144.015,Y -7.144,Z -8.549,A -90.000,B 90.000,C 0.000} C_DIS
LIN {X -48.031,Y -7.144,Z -8.549,A -90.000,B 90.000,C 0.000} C_DIS
LIN {X -46.688,Y -7.144,Z -8.853,A -90.000,B 90.000,C 0.000} C_DIS
LIN {X -45.339,Y -7.144,Z -9.133,A -90.000,B 90.000,C 0.000} C_DIS
LIN {X -43.986,Y -7.144,Z -9.390,A -90.000,B 90.000,C 0.000} C_DIS
LIN {X -39.168,Y -7.144,Z -10.232,A -90.000,B 90.000,C 0.000} C_DIS
LIN {X -34.361,Y -7.144,Z -11.134,A -90.000,B 90.000,C 0.000} C_DIS
LIN {X -29.565,Y -7.144,Z -12.094,A -90.000,B 90.000,C 0.000} C_DIS
LIN {X -24.781,Y -7.144,Z -13.113,A -90.000,B 90.000,C 0.000} C_DIS
LIN {X -20.010,Y -7.144,Z -14.191,A -90.000,B 90.000,C 0.000} C_DIS
LIN {X -15.253,Y -7.144,Z -15.327,A -90.000,B 90.000,C 0.000} C_DIS
LIN {X -12.563,Y -7.144,Z -16.098,A -90.000,B 90.000,C 0.000} C_DIS
LIN {X 144.015,Y -7.144,Z -16.098,A -90.000,B 90.000,C 0.000} C_DIS
LIN {X 144.015,Y -7.144,Z -23.646,A -90.000,B 90.000,C 0.000} C_DIS
LIN {X 17.296,Y -7.144,Z -23.646,A -90.000,B 90.000,C 0.000} C_DIS
LIN {X 19.189,Y -7.144,Z -24.083,A -90.000,B 90.000,C 0.000} C_DIS
LIN {X 21.079,Y -7.144,Z -24.531,A -90.000,B 90.000,C 0.000} C_DIS
LIN {X 23.253,Y -7.144,Z -24.892,A -90.000,B 90.000,C 0.000} C_DIS
LIN {X 25.416,Y -7.144,Z -25.315,A -90.000,B 90.000,C 0.000} C_DIS
LIN {X 27.566,Y -7.144,Z -25.798,A -90.000,B 90.000,C 0.000} C_DIS
LIN {X 29.701,Y -7.144,Z -26.343,A -90.000,B 90.000,C 0.000} C_DIS
LIN {X 31.820,Y -7.144,Z -26.948,A -90.000,B 90.000,C 0.000} C_DIS
LIN {X 33.921,Y -7.144,Z -27.613,A -90.000,B 90.000,C 0.000} C_DIS
LIN {X 37.450,Y -7.144,Z -28.776,A -90.000,B 90.000,C 0.000} C_DIS
LIN {X 40.989,Y -7.144,Z -29.909,A -90.000,B 90.000,C 0.000} C_DIS
LIN {X 43.116,Y -7.144,Z -30.535,A -90.000,B 90.000,C 0.000} C_DIS
LIN {X 45.233,Y -7.144,Z -31.195,A -90.000,B 90.000,C 0.000} C_DIS
LIN {X 98.289,Y -7.144,Z -31.195,A -90.000,B 90.000,C 0.000} C_DIS
LIN {X 96.315,Y -7.144,Z -32.157,A -90.000,B 90.000,C 0.000} C_DIS
LIN {X 94.368,Y -7.144,Z -33.171,A -90.000,B 90.000,C 0.000} C_DIS
LIN {X 92.448,Y -7.144,Z -34.238,A -90.000,B 90.000,C 0.000} C_DIS
LIN {X 90.558,Y -7.144,Z -35.355,A -90.000,B 90.000,C 0.000} C_DIS
LIN {X 88.699,Y -7.144,Z -36.523,A -90.000,B 90.000,C 0.000} C_DIS
LIN {X 87.662,Y -7.144,Z -37.232,A -90.000,B 90.000,C 0.000} C_DIS
LIN {X 86.648,Y -7.144,Z -37.973,A -90.000,B 90.000,C 0.000} C_DIS
LIN {X 85.657,Y -7.144,Z -38.744,A -90.000,B 90.000,C 0.000} C_DIS
LIN {X 63.604,Y -7.144,Z -38.744,A -90.000,B 90.000,C 0.000} C_DIS
LIN {X 66.273,Y -7.144,Z -40.150,A -90.000,B 90.000,C 0.000} C_DIS
LIN {X 68.913,Y -7.144,Z -41.609,A -90.000,B 90.000,C 0.000} C_DIS
LIN {X 71.524,Y -7.144,Z -43.119,A -90.000,B 90.000,C 0.000} C_DIS
LIN {X 74.105,Y -7.144,Z -44.681,A -90.000,B 90.000,C 0.000} C_DIS
LIN {X 76.654,Y -7.144,Z -46.293,A -90.000,B 90.000,C 0.000} C_DIS
LIN {X 78.397,Y -7.144,Z -46.293,A -90.000,B 90.000,C 0.000} C_DIS
LIN {X 79.365,Y -7.144,Z -45.038,A -90.000,B 90.000,C 0.000} C_DIS
LIN {X 80.382,Y -7.144,Z -43.821,A -90.000,B 90.000,C 0.000} C_DIS
LIN {X 81.444,Y -7.144,Z -42.644,A -90.000,B 90.000,C 0.000} C_DIS
LIN {X 82.551,Y -7.144,Z -41.509,A -90.000,B 90.000,C 0.000} C_DIS
LIN {X 83.702,Y -7.144,Z -40.418,A -90.000,B 90.000,C 0.000} C_DIS
LIN {X 84.894,Y -7.144,Z -39.373,A -90.000,B 90.000,C 0.000} C_DIS
LIN {X 86.125,Y -7.144,Z -38.374,A -90.000,B 90.000,C 0.000} C_DIS
LIN {X 87.394,Y -7.144,Z -37.423,A -90.000,B 90.000,C 0.000} C_DIS
LIN {X 88.699,Y -7.144,Z -36.523,A -90.000,B 90.000,C 0.000} C_DIS
LIN {X 90.540,Y -7.144,Z -35.366,A -90.000,B 90.000,C 0.000} C_DIS
LIN {X 92.411,Y -7.144,Z -34.259,A -90.000,B 90.000,C 0.000} C_DIS
LIN {X 94.312,Y -7.144,Z -33.202,A -90.000,B 90.000,C 0.000} C_DIS
LIN {X 96.239,Y -7.144,Z -32.196,A -90.000,B 90.000,C 0.000} C_DIS
LIN {X 98.192,Y -7.144,Z -31.241,A -90.000,B 90.000,C 0.000} C_DIS
LIN {X 100.170,Y -7.144,Z -30.338,A -90.000,B 90.000,C 0.000} C_DIS
LIN {X 102.172,Y -7.144,Z -29.488,A -90.000,B 90.000,C 0.000} C_DIS
LIN {X 104.195,Y -7.144,Z -28.692,A -90.000,B 90.000,C 0.000} C_DIS
LIN {X 105.149,Y -7.144,Z -28.311,A -90.000,B 90.000,C 0.000} C_DIS
LIN {X 106.126,Y -7.144,Z -27.993,A -90.000,B 90.000,C 0.000} C_DIS
LIN {X 107.123,Y -7.144,Z -27.742,A -90.000,B 90.000,C 0.000} C_DIS
LIN {X 108.133,Y -7.144,Z -27.557,A -90.000,B 90.000,C 0.000} C_DIS
LIN {X 109.154,Y -7.144,Z -27.440,A -90.000,B 90.000,C 0.000} C_DIS
LIN {X 110.180,Y -7.144,Z -27.391,A -90.000,B 90.000,C 0.000} C_DIS
LIN {X 111.208,Y -7.144,Z -27.410,A -90.000,B 90.000,C 0.000} C_DIS
LIN {X 112.231,Y -7.144,Z -27.498,A -90.000,B 90.000,C 0.000} C_DIS
LIN {X 113.247,Y -7.144,Z -27.653,A -90.000,B 90.000,C 0.000} C_DIS
LIN {X 114.250,Y -7.144,Z -27.876,A -90.000,B 90.000,C 0.000} C_DIS
LIN {X 115.236,Y -7.144,Z -28.165,A -90.000,B 90.000,C 0.000} C_DIS
LIN {X 116.201,Y -7.144,Z -28.518,A -90.000,B 90.000,C 0.000} C_DIS
LIN {X 117.140,Y -7.144,Z -28.935,A -90.000,B 90.000,C 0.000} C_DIS
LIN {X 118.049,Y -7.144,Z -29.414,A -90.000,B 90.000,C 0.000} C_DIS
LIN {X 118.924,Y -7.144,Z -29.951,A -90.000,B 90.000,C 0.000} C_DIS
LIN {X 119.762,Y -7.144,Z -30.546,A -90.000,B 90.000,C 0.000} C_DIS
LIN {X 120.559,Y -7.144,Z -31.195,A -90.000,B 90.000,C 0.000} C_DIS
LIN {X 144.015,Y -7.144,Z -31.195,A -90.000,B 90.000,C 0.000} C_DIS
LIN {X 144.015,Y -7.144,Z -38.744,A -90.000,B 90.000,C 0.000} C_DIS
LIN {X 124.956,Y -7.144,Z -38.744,A -90.000,B 90.000,C 0.000} C_DIS
LIN {X 125.148,Y -7.144,Z -39.640,A -90.000,B 90.000,C 0.000} C_DIS
LIN {X 125.291,Y -7.144,Z -40.545,A -90.000,B 90.000,C 0.000} C_DIS
LIN {X 125.384,Y -7.144,Z -41.456,A -90.000,B 90.000,C 0.000} C_DIS
LIN {X 125.427,Y -7.144,Z -42.371,A -90.000,B 90.000,C 0.000} C_DIS
LIN {X 125.420,Y -7.144,Z -43.288,A -90.000,B 90.000,C 0.000} C_DIS
LIN {X 125.363,Y -7.144,Z -44.202,A -90.000,B 90.000,C 0.000} C_DIS
LIN {X 125.205,Y -7.144,Z -45.251,A -90.000,B 90.000,C 0.000} C_DIS
LIN {X 125.008,Y -7.144,Z -46.293,A -90.000,B 90.000,C 0.000} C_DIS
LIN {X 144.015,Y -7.144,Z -46.293,A -90.000,B 90.000,C 0.000} C_DIS
LIN {X 144.015,Y -7.144,Z -53.842,A -90.000,B 90.000,C 0.000} C_DIS
LIN {X 122.298,Y -7.144,Z -53.842,A -90.000,B 90.000,C 0.000} C_DIS
